LIN {X -0.062,Y -576.577,Z 1331.562,A 0.000,B 0.000,C 90.000,E1 137.229} C_DIS
LIN {X -0.112,Y -582.728,Z 1331.561,A 0.000,B 0.000,C 90.000,E1 136.905} C_DIS
LIN {X -0.019,Y -586.967,Z 1331.559,A 0.000,B 0.000,C 90.000,E1 136.620} C_DIS
LIN {X -0.228,Y -592.649,Z 1331.557,A 0.000,B 0.000,C 90.000,E1 136.215} C_DIS
LIN {X -0.386,Y -596.705,Z 1331.555,A 0.000,B 0.000,C 90.000,E1 135.891} C_DIS
LIN {X 0.112,Y -600.626,Z 1331.553,A 0.000,B 0.000,C 90.000,E1 135.486} C_DIS
LIN {X -0.001,Y -606.973,Z 1331.549,A 0.000,B 0.000,C 90.000,E1 134.879} C_DIS
LIN {X -0.167,Y -610.638,Z 1331.547,A 0.000,B 0.000,C 90.000,E1 134.514} C_DIS
LIN {X -0.298,Y -618.235,Z 1331.542,A 0.000,B 0.000,C 90.000,E1 133.623} C_DIS
LIN {X -0.305,Y -624.374,Z 1331.538,A 0.000,B 0.000,C 90.000,E1 132.852} C_DIS
LIN {X -0.246,Y -630.021,Z 1331.534,A 0.000,B 0.000,C 90.000,E1 132.081} C_DIS
LIN {X -0.360,Y -639.806,Z 1331.526,A 0.000,B 0.000,C 90.000,E1 130.701} C_DIS
LIN {X -0.233,Y -647.239,Z 1331.520,A 0.000,B 0.000,C 90.000,E1 129.564} C_DIS
LIN {X 0.131,Y -651.204,Z 1331.516,A 0.000,B 0.000,C 90.000,E1 128.910} C_DIS
LIN {X 0.016,Y -657.983,Z 1331.510,A 0.000,B 0.000,C 90.000,E1 127.810} C_DIS
LIN {X -0.050,Y -661.508,Z 1331.507,A 0.000,B 0.000,C 90.000,E1 127.202} C_DIS
LIN {X 0.091,Y -665.436,Z 1331.503,A 0.000,B 0.000,C 90.000,E1 126.457} C_DIS
LIN {X -0.320,Y -668.389,Z 1331.499,A 0.000,B 0.000,C 90.000,E1 125.884} C_DIS
LIN {X 0.287,Y -671.652,Z 1331.495,A 0.000,B 0.000,C 90.000,E1 125.105} C_DIS
LIN {X -0.155,Y -673.656,Z 1331.493,A 0.000,B 0.000,C 90.000,E1 124.659} C_DIS
LIN {X 0.118,Y -676.353,Z 1331.489,A 0.000,B 0.000,C 90.000,E1 123.913} C_DIS
LIN {X -0.143,Y -678.675,Z 1331.484,A 0.000,B 0.000,C 90.000,E1 123.214} C_DIS
LIN {X -0.205,Y -681.301,Z 1331.479,A 0.000,B 0.000,C 90.000,E1 122.260} C_DIS
LIN {X -0.208,Y -683.012,Z 1331.475,A 0.000,B 0.000,C 90.000,E1 121.544} C_DIS
LIN {X 0.166,Y -684.515,Z 1331.471,A 0.000,B 0.000,C 90.000,E1 120.797} C_DIS
LIN {X 0.207,Y -685.843,Z 1331.467,A 0.000,B 0.000,C 90.000,E1 120.079} C_DIS
LIN {X -0.333,Y -686.828,Z 1331.463,A 0.000,B 0.000,C 90.000,E1 119.411} C_DIS
LIN {X -0.267,Y -687.514,Z 1331.459,A 0.000,B 0.000,C 90.000,E1 118.693} C_DIS
LIN {X -0.193,Y -687.911,Z 1331.455,A 0.000,B 0.000,C 90.000,E1 117.975} C_DIS
LIN {X 0.110,Y -688.126,Z 1331.450,A 0.000,B 0.000,C 90.000,E1 117.001} C_DIS
LIN {X -0.124,Y -688.029,Z 1331.446,A 0.000,B 0.000,C 90.000,E1 116.309} C_DIS
LIN {X -0.282,Y -687.859,Z 1331.443,A 0.000,B 0.000,C 90.000,E1 115.848} C_DIS
LIN {X 0.173,Y -687.510,Z 1331.441,A 0.000,B 0.000,C 90.000,E1 115.335} C_DIS
LIN {X -0.064,Y -686.536,Z 1331.437,A 0.000,B 0.000,C 90.000,E1 114.643} C_DIS
LIN {X 0.097,Y -685.440,Z 1331.434,A 0.000,B 0.000,C 90.000,E1 114.155} C_DIS
LIN {X -0.309,Y -684.576,Z 1331.433,A 0.000,B 0.000,C 90.000,E1 113.951} C_DIS
LIN {X -0.155,Y -682.367,Z 1331.430,A 0.000,B 0.000,C 90.000,E1 113.462} C_DIS
LIN {X -0.051,Y -681.471,Z 1331.430,A 0.000,B 0.000,C 90.000,E1 113.334} C_DIS
LIN {X 0.357,Y -676.839,Z 1331.427,A 0.000,B 0.000,C 90.000,E1 112.823} C_DIS
LIN {X 0.189,Y -675.138,Z 1331.426,A 0.000,B 0.000,C 90.000,E1 112.717} C_DIS
LIN {X -0.013,Y -668.323,Z 1331.425,A 0.000,B 0.000,C 90.000,E1 112.408} C_DIS
LIN {X -0.068,Y -666.391,Z 1331.424,A 0.000,B 0.000,C 90.000,E1 112.333} C_DIS
LIN {X 0.000,Y -659.861,Z 1331.423,A 0.000,B 0.000,C 90.000,E1 112.153} C_DIS
LIN {X 0.072,Y -657.595,Z 1331.423,A 0.000,B 0.000,C 90.000,E1 112.099} C_DIS
LIN {X -0.013,Y -646.608,Z 1331.422,A 0.000,B 0.000,C 90.000,E1 111.950} C_DIS
LIN {X 0.023,Y -643.350,Z 1331.422,A 0.000,B 0.000,C 90.000,E1 111.897} C_DIS
LIN {X 0.052,Y -641.499,Z 1331.421,A 0.000,B 0.000,C 90.000,E1 111.844} C_DIS
LIN {X 0.018,Y -641.457,Z 1331.421,A 0.000,B 0.000,C 90.000,E1 111.844} C_DIS
LIN {X -0.197,Y -642.666,Z 1331.420,A 0.000,B 0.000,C 90.000,E1 111.663} C_DIS
LIN {X 0.238,Y -647.960,Z 1331.417,A 0.000,B 0.000,C 90.000,E1 110.972} C_DIS
LIN {X 0.157,Y -651.763,Z 1331.414,A 0.000,B 0.000,C 90.000,E1 110.482} C_DIS
LIN {X -0.079,Y -655.885,Z 1331.411,A 0.000,B 0.000,C 90.000,E1 109.885} C_DIS
LIN {X -0.057,Y -659.444,Z 1331.407,A 0.000,B 0.000,C 90.000,E1 109.268} C_DIS
LIN {X -0.226,Y -662.475,Z 1331.404,A 0.000,B 0.000,C 90.000,E1 108.671} C_DIS
LIN {X -0.313,Y -665.638,Z 1331.400,A 0.000,B 0.000,C 90.000,E1 107.946} C_DIS
LIN {X -0.373,Y -668.406,Z 1331.396,A 0.000,B 0.000,C 90.000,E1 107.221} C_DIS
LIN {X 0.306,Y -670.155,Z 1331.393,A 0.000,B 0.000,C 90.000,E1 106.677} C_DIS
LIN {X 0.098,Y -672.322,Z 1331.389,A 0.000,B 0.000,C 90.000,E1 105.969} C_DIS
LIN {X 0.155,Y -673.642,Z 1331.386,A 0.000,B 0.000,C 90.000,E1 105.481} C_DIS
LIN {X -0.019,Y -675.326,Z 1331.382,A 0.000,B 0.000,C 90.000,E1 104.773} C_DIS
LIN {X -0.124,Y -676.313,Z 1331.379,A 0.000,B 0.000,C 90.000,E1 104.300} C_DIS
LIN {X -0.270,Y -677.357,Z 1331.375,A 0.000,B 0.000,C 90.000,E1 103.592} C_DIS
LIN {X 0.299,Y -677.875,Z 1331.373,A 0.000,B 0.000,C 90.000,E1 103.063} C_DIS
LIN {X 0.121,Y -678.259,Z 1331.367,A 0.000,B 0.000,C 90.000,E1 102.119} C_DIS
LIN {X -0.151,Y -678.121,Z 1331.363,A 0.000,B 0.000,C 90.000,E1 101.422} C_DIS
LIN {X -0.243,Y -677.718,Z 1331.361,A 0.000,B 0.000,C 90.000,E1 100.950} C_DIS
LIN {X 0.152,Y -676.717,Z 1331.357,A 0.000,B 0.000,C 90.000,E1 100.197} C_DIS
LIN {X 0.045,Y -675.836,Z 1331.354,A 0.000,B 0.000,C 90.000,E1 99.726} C_DIS
LIN {X -0.183,Y -674.676,Z 1331.351,A 0.000,B 0.000,C 90.000,E1 99.265} C_DIS
LIN {X 0.251,Y -673.113,Z 1331.349,A 0.000,B 0.000,C 90.000,E1 98.746} C_DIS
LIN {X -0.061,Y -670.258,Z 1331.345,A 0.000,B 0.000,C 90.000,E1 98.049} C_DIS
LIN {X -0.313,Y -668.104,Z 1331.342,A 0.000,B 0.000,C 90.000,E1 97.587} C_DIS
LIN {X -0.107,Y -663.890,Z 1331.337,A 0.000,B 0.000,C 90.000,E1 96.720} C_DIS
LIN {X 0.135,Y -659.920,Z 1331.333,A 0.000,B 0.000,C 90.000,E1 95.967} C_DIS
LIN {X -0.253,Y -656.964,Z 1331.331,A 0.000,B 0.000,C 90.000,E1 95.511} C_DIS
LIN {X -0.039,Y -652.848,Z 1331.327,A 0.000,B 0.000,C 90.000,E1 94.878} C_DIS
LIN {X 0.135,Y -648.411,Z 1331.324,A 0.000,B 0.000,C 90.000,E1 94.245} C_DIS
LIN {X -0.262,Y -644.634,Z 1331.321,A 0.000,B 0.000,C 90.000,E1 93.784} C_DIS
LIN {X 0.038,Y -641.655,Z 1331.319,A 0.000,B 0.000,C 90.000,E1 93.383} C_DIS
LIN {X 0.109,Y -636.035,Z 1331.315,A 0.000,B 0.000,C 90.000,E1 92.751} C_DIS
LIN {X 0.212,Y -629.898,Z 1331.312,A 0.000,B 0.000,C 90.000,E1 92.121} C_DIS
LIN {X 0.185,Y -619.842,Z 1331.307,A 0.000,B 0.000,C 90.000,E1 91.146} C_DIS
LIN {X -0.039,Y -615.737,Z 1331.304,A 0.000,B 0.000,C 90.000,E1 90.802} C_DIS
LIN {X -0.001,Y -610.127,Z 1331.302,A 0.000,B 0.000,C 90.000,E1 90.344} C_DIS
LIN {X 0.018,Y -608.545,Z 1331.301,A 0.000,B 0.000,C 90.000,E1 90.229} C_DIS
LIN {X 0.053,Y -602.004,Z 1331.299,A 0.000,B 0.000,C 90.000,E1 89.828} C_DIS
LIN {X -0.038,Y -594.968,Z 1331.297,A 0.000,B 0.000,C 90.000,E1 89.484} C_DIS
LIN {X -0.226,Y -587.786,Z 1331.296,A 0.000,B 0.000,C 90.000,E1 89.198} C_DIS
LIN {X -0.262,Y -577.938,Z 1331.293,A 0.000,B 0.000,C 90.000,E1 88.797} C_DIS
LIN {X 0.160,Y -576.610,Z 1331.293,A 0.000,B 0.000,C 90.000,E1 88.682} C_DIS
LIN {X 0.074,Y -573.479,Z 1331.292,A 0.000,B 0.000,C 90.000,E1 88.453} C_DIS
LIN {X 0.131,Y -573.050,Z 1331.291,A 0.000,B 0.000,C 90.000,E1 88.396} C_DIS
LIN {X 0.097,Y -573.038,Z 1331.291,A 0.000,B 0.000,C 90.000,E1 88.396} C_DIS
LIN {X 0.284,Y -572.281,Z 1331.290,A 0.000,B 0.000,C 90.000,E1 88.108} C_DIS
LIN {X 0.249,Y -572.134,Z 1331.287,A 0.000,B 0.000,C 90.000,E1 87.650} C_DIS
LIN {X 0.140,Y -574.875,Z 1331.271,A 0.000,B 0.000,C 90.000,E1 84.666} C_DIS
LIN {X -0.183,Y -577.423,Z 1331.258,A 0.000,B 0.000,C 90.000,E1 82.527} C_DIS
LIN {X -0.207,Y -579.382,Z 1331.249,A 0.000,B 0.000,C 90.000,E1 80.905} C_DIS
LIN {X -0.097,Y -581.262,Z 1331.240,A 0.000,B 0.000,C 90.000,E1 79.275} C_DIS
LIN {X -0.192,Y -582.690,Z 1331.233,A 0.000,B 0.000,C 90.000,E1 77.937} C_DIS
LIN {X 0.084,Y -584.057,Z 1331.224,A 0.000,B 0.000,C 90.000,E1 76.297} C_DIS
LIN {X 0.042,Y -584.865,Z 1331.218,A 0.000,B 0.000,C 90.000,E1 75.227} C_DIS
LIN {X -0.233,Y -586.188,Z 1331.208,A 0.000,B 0.000,C 90.000,E1 73.378} C_DIS
LIN {X -0.160,Y -587.169,Z 1331.199,A 0.000,B 0.000,C 90.000,E1 71.764} C_DIS
LIN {X 0.106,Y -588.256,Z 1331.190,A 0.000,B 0.000,C 90.000,E1 70.134} C_DIS
LIN {X -0.197,Y -589.629,Z 1331.178,A 0.000,B 0.000,C 90.000,E1 68.028} C_DIS
LIN {X 0.088,Y -591.002,Z 1331.166,A 0.000,B 0.000,C 90.000,E1 65.869} C_DIS
LIN {X 0.208,Y -591.781,Z 1331.160,A 0.000,B 0.000,C 90.000,E1 64.793} C_DIS
LIN {X 0.044,Y -593.113,Z 1331.150,A 0.000,B 0.000,C 90.000,E1 62.948} C_DIS
LIN {X -0.060,Y -594.629,Z 1331.140,A 0.000,B 0.000,C 90.000,E1 61.101} C_DIS
LIN {X -0.108,Y -596.409,Z 1331.129,A 0.000,B 0.000,C 90.000,E1 59.253} C_DIS
LIN {X 0.188,Y -598.296,Z 1331.119,A 0.000,B 0.000,C 90.000,E1 57.375} C_DIS
LIN {X -0.133,Y -599.720,Z 1331.112,A 0.000,B 0.000,C 90.000,E1 56.087} C_DIS
LIN {X -0.101,Y -601.081,Z 1331.104,A 0.000,B 0.000,C 90.000,E1 54.769} C_DIS
LIN {X 0.216,Y -603.046,Z 1331.093,A 0.000,B 0.000,C 90.000,E1 52.637} C_DIS
LIN {X 0.171,Y -603.992,Z 1331.085,A 0.000,B 0.000,C 90.000,E1 51.331} C_DIS
LIN {X 0.058,Y -604.891,Z 1331.078,A 0.000,B 0.000,C 90.000,E1 50.033} C_DIS
LIN {X -0.225,Y -605.436,Z 1331.072,A 0.000,B 0.000,C 90.000,E1 49.013} C_DIS
LIN {X -0.114,Y -605.758,Z 1331.066,A 0.000,B 0.000,C 90.000,E1 47.957} C_DIS
LIN {X -0.176,Y -606.045,Z 1331.056,A 0.000,B 0.000,C 90.000,E1 46.134} C_DIS
LIN {X -0.084,Y -606.096,Z 1331.050,A 0.000,B 0.000,C 90.000,E1 45.081} C_DIS
LIN {X 0.008,Y -605.920,Z 1331.045,A 0.000,B 0.000,C 90.000,E1 44.028} C_DIS
LIN {X -0.130,Y -605.679,Z 1331.040,A 0.000,B 0.000,C 90.000,E1 43.257} C_DIS
LIN {X 0.198,Y -605.220,Z 1331.033,A 0.000,B 0.000,C 90.000,E1 41.919} C_DIS
LIN {X -0.094,Y -604.592,Z 1331.024,A 0.000,B 0.000,C 90.000,E1 40.378} C_DIS
LIN {X -0.332,Y -603.783,Z 1331.016,A 0.000,B 0.000,C 90.000,E1 38.830} C_DIS
LIN {X -0.033,Y -603.330,Z 1331.011,A 0.000,B 0.000,C 90.000,E1 38.016} C_DIS
LIN {X 0.147,Y -602.529,Z 1331.005,A 0.000,B 0.000,C 90.000,E1 36.950} C_DIS
LIN {X -0.168,Y -601.163,Z 1331.000,A 0.000,B 0.000,C 90.000,E1 35.931} C_DIS
LIN {X 0.225,Y -599.928,Z 1330.995,A 0.000,B 0.000,C 90.000,E1 35.105} C_DIS
LIN {X 0.016,Y -598.152,Z 1330.989,A 0.000,B 0.000,C 90.000,E1 34.072} C_DIS
LIN {X -0.344,Y -597.115,Z 1330.986,A 0.000,B 0.000,C 90.000,E1 33.579} C_DIS
LIN {X 0.127,Y -594.080,Z 1330.979,A 0.000,B 0.000,C 90.000,E1 32.212} C_DIS
LIN {X 0.237,Y -592.668,Z 1330.976,A 0.000,B 0.000,C 90.000,E1 31.671} C_DIS
LIN {X -0.388,Y -589.347,Z 1330.970,A 0.000,B 0.000,C 90.000,E1 30.669} C_DIS
LIN {X 0.082,Y -586.485,Z 1330.966,A 0.000,B 0.000,C 90.000,E1 29.823} C_DIS
LIN {X 0.135,Y -584.367,Z 1330.963,A 0.000,B 0.000,C 90.000,E1 29.283} C_DIS
LIN {X 0.039,Y -580.809,Z 1330.958,A 0.000,B 0.000,C 90.000,E1 28.487} C_DIS
LIN {X -0.228,Y -578.276,Z 1330.955,A 0.000,B 0.000,C 90.000,E1 27.975} C_DIS
LIN {X 0.112,Y -574.080,Z 1330.951,A 0.000,B 0.000,C 90.000,E1 27.129} C_DIS
LIN {X -0.283,Y -570.240,Z 1330.947,A 0.000,B 0.000,C 90.000,E1 26.488} C_DIS
LIN {X -0.196,Y -566.070,Z 1330.943,A 0.000,B 0.000,C 90.000,E1 25.796} C_DIS
LIN {X 0.191,Y -562.510,Z 1330.940,A 0.000,B 0.000,C 90.000,E1 25.207} C_DIS
LIN {X 0.307,Y -558.636,Z 1330.937,A 0.000,B 0.000,C 90.000,E1 24.643} C_DIS
LIN {X 0.062,Y -551.462,Z 1330.932,A 0.000,B 0.000,C 90.000,E1 23.695} C_DIS
LIN {X 0.143,Y -544.586,Z 1330.927,A 0.000,B 0.000,C 90.000,E1 22.845} C_DIS
LIN {X -0.216,Y -538.717,Z 1330.923,A 0.000,B 0.000,C 90.000,E1 22.206} C_DIS
LIN {X 0.226,Y -533.817,Z 1330.920,A 0.000,B 0.000,C 90.000,E1 21.589} C_DIS
LIN {X 0.072,Y -523.295,Z 1330.914,A 0.000,B 0.000,C 90.000,E1 20.482} C_DIS
LIN {X -0.222,Y -512.601,Z 1330.908,A 0.000,B 0.000,C 90.000,E1 19.396} C_DIS
LIN {X 0.248,Y -503.297,Z 1330.902,A 0.000,B 0.000,C 90.000,E1 18.362} C_DIS
LIN {X 0.005,Y -492.422,Z 1330.896,A 0.000,B 0.000,C 90.000,E1 17.330} C_DIS
LIN {X 0.045,Y -478.128,Z 1330.889,A 0.000,B 0.000,C 90.000,E1 15.969} C_DIS
LIN {X 0.080,Y -468.016,Z 1330.884,A 0.000,B 0.000,C 90.000,E1 15.009} C_DIS
LIN {X 0.147,Y -451.951,Z 1330.875,A 0.000,B 0.000,C 90.000,E1 13.480} C_DIS
LIN {X -0.018,Y -431.896,Z 1330.864,A 0.000,B 0.000,C 90.000,E1 11.478} C_DIS
LIN {X -0.191,Y -417.628,Z 1330.855,A 0.000,B 0.000,C 90.000,E1 9.962} C_DIS
LIN {X -0.042,Y -404.851,Z 1330.847,A 0.000,B 0.000,C 90.000,E1 8.511} C_DIS
LIN {X -0.076,Y -399.255,Z 1330.844,A 0.000,B 0.000,C 90.000,E1 7.871} C_DIS
LIN {X -0.072,Y -395.398,Z 1330.841,A 0.000,B 0.000,C 90.000,E1 7.352} C_DIS
LIN {X 0.017,Y -395.218,Z 1330.841,A 0.000,B 0.000,C 90.000,E1 7.296} C_DIS
LIN {X -0.020,Y -395.210,Z 1330.841,A 0.000,B 0.000,C 90.000,E1 7.296} C_DIS
LIN {X 0.119,Y -395.467,Z 1330.840,A 0.000,B 0.000,C 90.000,E1 7.182} C_DIS
LIN {X 0.081,Y -395.514,Z 1330.840,A 0.000,B 0.000,C 90.000,E1 7.182} C_DIS
LIN {X 0.073,Y -398.573,Z 1330.838,A 0.000,B 0.000,C 90.000,E1 6.891} C_DIS
LIN {X -0.153,Y -400.282,Z 1330.838,A 0.000,B 0.000,C 90.000,E1 6.777} C_DIS
LIN {X 0.049,Y -413.967,Z 1330.833,A 0.000,B 0.000,C 90.000,E1 5.853} C_DIS
LIN {X 0.107,Y -417.244,Z 1330.831,A 0.000,B 0.000,C 90.000,E1 5.625} C_DIS
LIN {X -0.069,Y -425.051,Z 1330.828,A 0.000,B 0.000,C 90.000,E1 5.049} C_DIS
LIN {X 0.062,Y -429.652,Z 1330.826,A 0.000,B 0.000,C 90.000,E1 4.645} C_DIS
LIN {X -0.137,Y -438.664,Z 1330.821,A 0.000,B 0.000,C 90.000,E1 3.841} C_DIS
LIN {X 0.072,Y -445.876,Z 1330.817,A 0.000,B 0.000,C 90.000,E1 3.094} C_DIS
LIN {X 0.057,Y -452.935,Z 1330.813,A 0.000,B 0.000,C 90.000,E1 2.350} C_DIS
LIN {X -0.061,Y -459.618,Z 1330.809,A 0.000,B 0.000,C 90.000,E1 1.604} C_DIS
LIN {X 0.202,Y -465.898,Z 1330.805,A 0.000,B 0.000,C 90.000,E1 0.802} C_DIS
LIN {X 0.191,Y -470.762,Z 1330.801,A 0.000,B 0.000,C 90.000,E1 0.172} C_DIS
LIN {X 0.093,Y -476.831,Z 1330.796,A 0.000,B 0.000,C 90.000,E1 359.312} C_DIS
LIN {X -0.177,Y -481.811,Z 1330.792,A 0.000,B 0.000,C 90.000,E1 358.568} C_DIS
LIN {X 0.100,Y -486.338,Z 1330.788,A 0.000,B 0.000,C 90.000,E1 357.764} C_DIS
LIN {X -0.087,Y -490.693,Z 1330.783,A 0.000,B 0.000,C 90.000,E1 357.020} C_DIS
LIN {X 0.112,Y -493.901,Z 1330.780,A 0.000,B 0.000,C 90.000,E1 356.388} C_DIS
LIN {X 0.022,Y -497.559,Z 1330.776,A 0.000,B 0.000,C 90.000,E1 355.641} C_DIS
LIN {X 0.146,Y -501.640,Z 1330.771,A 0.000,B 0.000,C 90.000,E1 354.723} C_DIS
LIN {X 0.123,Y -504.809,Z 1330.767,A 0.000,B 0.000,C 90.000,E1 353.976} C_DIS
LIN {X -0.010,Y -507.132,Z 1330.763,A 0.000,B 0.000,C 90.000,E1 353.394} C_DIS
LIN {X 0.157,Y -511.513,Z 1330.757,A 0.000,B 0.000,C 90.000,E1 352.186} C_DIS
LIN {X 0.081,Y -513.454,Z 1330.753,A 0.000,B 0.000,C 90.000,E1 351.602} C_DIS
LIN {X -0.100,Y -516.862,Z 1330.747,A 0.000,B 0.000,C 90.000,E1 350.443} C_DIS
LIN {X -0.138,Y -519.199,Z 1330.742,A 0.000,B 0.000,C 90.000,E1 349.567} C_DIS
LIN {X -0.249,Y -521.216,Z 1330.737,A 0.000,B 0.000,C 90.000,E1 348.701} C_DIS
LIN {X -0.133,Y -523.042,Z 1330.732,A 0.000,B 0.000,C 90.000,E1 347.813} C_DIS
LIN {X -0.090,Y -525.127,Z 1330.726,A 0.000,B 0.000,C 90.000,E1 346.645} C_DIS
LIN {X -0.062,Y -526.045,Z 1330.723,A 0.000,B 0.000,C 90.000,E1 346.061} C_DIS
LIN {X 0.117,Y -527.163,Z 1330.718,A 0.000,B 0.000,C 90.000,E1 345.172} C_DIS
LIN {X -0.198,Y -528.147,Z 1330.713,A 0.000,B 0.000,C 90.000,E1 344.338} C_DIS
LIN {X 0.004,Y -528.829,Z 1330.708,A 0.000,B 0.000,C 90.000,E1 343.449} C_DIS
LIN {X 0.192,Y -529.155,Z 1330.705,A 0.000,B 0.000,C 90.000,E1 342.851} C_DIS
LIN {X 0.068,Y -529.356,Z 1330.698,A 0.000,B 0.000,C 90.000,E1 341.710} C_DIS
LIN {X -0.065,Y -529.297,Z 1330.694,A 0.000,B 0.000,C 90.000,E1 340.859} C_DIS
LIN {X 0.300,Y -528.995,Z 1330.690,A 0.000,B 0.000,C 90.000,E1 340.242} C_DIS
LIN {X -0.145,Y -528.127,Z 1330.684,A 0.000,B 0.000,C 90.000,E1 339.135} C_DIS
LIN {X 0.203,Y -526.930,Z 1330.679,A 0.000,B 0.000,C 90.000,E1 338.230} C_DIS
LIN {X 0.093,Y -524.425,Z 1330.671,A 0.000,B 0.000,C 90.000,E1 336.794} C_DIS
LIN {X 0.103,Y -522.563,Z 1330.666,A 0.000,B 0.000,C 90.000,E1 335.921} C_DIS
LIN {X 0.089,Y -520.368,Z 1330.661,A 0.000,B 0.000,C 90.000,E1 335.049} C_DIS
LIN {X -0.061,Y -516.851,Z 1330.655,A 0.000,B 0.000,C 90.000,E1 333.896} C_DIS
LIN {X 0.090,Y -512.241,Z 1330.647,A 0.000,B 0.000,C 90.000,E1 332.410} C_DIS
LIN {X 0.182,Y -509.383,Z 1330.642,A 0.000,B 0.000,C 90.000,E1 331.513} C_DIS
LIN {X -0.028,Y -506.591,Z 1330.638,A 0.000,B 0.000,C 90.000,E1 330.795} C_DIS
LIN {X 0.109,Y -504.527,Z 1330.635,A 0.000,B 0.000,C 90.000,E1 330.333} C_DIS
LIN {X -0.014,Y -502.929,Z 1330.634,A 0.000,B 0.000,C 90.000,E1 330.049} C_DIS
LIN {X 0.041,Y -500.988,Z 1330.632,A 0.000,B 0.000,C 90.000,E1 329.744} C_DIS
LIN {X -0.151,Y -499.776,Z 1330.631,A 0.000,B 0.000,C 90.000,E1 329.616} C_DIS
LIN {X -0.090,Y -498.041,Z 1330.630,A 0.000,B 0.000,C 90.000,E1 329.459} C_DIS
LIN {X -0.222,Y -472.486,Z 1330.620,A 0.000,B 0.000,C 90.000,E1 327.661} C_DIS
LIN {X -0.018,Y -449.591,Z 1330.610,A 0.000,B 0.000,C 90.000,E1 325.801} C_DIS
LIN {X 0.050,Y -428.701,Z 1330.600,A 0.000,B 0.000,C 90.000,E1 323.909} C_DIS
LIN {X 0.168,Y -408.338,Z 1330.588,A 0.000,B 0.000,C 90.000,E1 321.823} C_DIS
LIN {X -0.045,Y -389.975,Z 1330.576,A 0.000,B 0.000,C 90.000,E1 319.747} C_DIS
LIN {X 0.005,Y -377.260,Z 1330.567,A 0.000,B 0.000,C 90.000,E1 318.119} C_DIS
LIN {X 0.219,Y -377.263,Z 1330.567,A 0.000,B 0.000,C 90.000,E1 318.081} C_DIS
LIN {X -0.089,Y -377.906,Z 1330.565,A 0.000,B 0.000,C 90.000,E1 317.634} C_DIS
LIN {X -0.082,Y -378.509,Z 1330.561,A 0.000,B 0.000,C 90.000,E1 316.905} C_DIS
LIN {X 0.218,Y -384.511,Z 1330.528,A 0.000,B 0.000,C 90.000,E1 311.067} C_DIS
LIN {X -0.029,Y -384.928,Z 1330.526,A 0.000,B 0.000,C 90.000,E1 310.744} C_DIS
LIN {X -0.109,Y -390.684,Z 1330.495,A 0.000,B 0.000,C 90.000,E1 305.025} C_DIS
LIN {X -0.042,Y -391.181,Z 1330.493,A 0.000,B 0.000,C 90.000,E1 304.659} C_DIS
LIN {X 0.086,Y -396.896,Z 1330.459,A 0.000,B 0.000,C 90.000,E1 298.615} C_DIS
LIN {X -0.137,Y -397.492,Z 1330.453,A 0.000,B 0.000,C 90.000,E1 297.590} C_DIS
LIN {X 0.096,Y -401.633,Z 1330.426,A 0.000,B 0.000,C 90.000,E1 292.642} C_DIS
LIN {X -0.153,Y -404.705,Z 1330.395,A 0.000,B 0.000,C 90.000,E1 287.094} C_DIS
LIN {X -0.161,Y -406.131,Z 1330.364,A 0.000,B 0.000,C 90.000,E1 281.535} C_DIS
LIN {X -0.118,Y -405.722,Z 1330.356,A 0.000,B 0.000,C 90.000,E1 280.141} C_DIS
LIN {X -0.068,Y -405.689,Z 1330.333,A 0.000,B 0.000,C 90.000,E1 275.967} C_DIS
LIN {X -0.031,Y -403.464,Z 1330.304,A 0.000,B 0.000,C 90.000,E1 270.745} C_DIS
LIN {X -0.063,Y -403.248,Z 1330.302,A 0.000,B 0.000,C 90.000,E1 270.401} C_DIS
LIN {X 0.116,Y -398.868,Z 1330.271,A 0.000,B 0.000,C 90.000,E1 264.780} C_DIS
LIN {X 0.014,Y -393.344,Z 1330.244,A 0.000,B 0.000,C 90.000,E1 259.859} C_DIS
LIN {X -0.064,Y -392.771,Z 1330.240,A 0.000,B 0.000,C 90.000,E1 259.162} C_DIS
LIN {X 0.015,Y -386.319,Z 1330.214,A 0.000,B 0.000,C 90.000,E1 254.519} C_DIS
LIN {X -0.024,Y -385.215,Z 1330.208,A 0.000,B 0.000,C 90.000,E1 253.449} C_DIS
LIN {X 0.017,Y -384.010,Z 1330.204,A 0.000,B 0.000,C 90.000,E1 252.725} C_DIS
LIN {X -0.154,Y -377.445,Z 1330.180,A 0.000,B 0.000,C 90.000,E1 248.411} C_DIS
LIN {X -0.062,Y -376.171,Z 1330.174,A 0.000,B 0.000,C 90.000,E1 247.305} C_DIS
LIN {X -0.073,Y -368.341,Z 1330.147,A 0.000,B 0.000,C 90.000,E1 242.538} C_DIS
LIN {X -0.030,Y -366.478,Z 1330.139,A 0.000,B 0.000,C 90.000,E1 241.051} C_DIS
LIN {X 0.055,Y -365.937,Z 1330.137,A 0.000,B 0.000,C 90.000,E1 240.667} C_DIS
LIN {X -0.055,Y -359.116,Z 1330.114,A 0.000,B 0.000,C 90.000,E1 236.580} C_DIS
LIN {X -0.059,Y -356.258,Z 1330.102,A 0.000,B 0.000,C 90.000,E1 234.322} C_DIS
LIN {X 0.161,Y -355.737,Z 1330.100,A 0.000,B 0.000,C 90.000,E1 233.909} C_DIS
LIN {X -0.036,Y -348.721,Z 1330.074,A 0.000,B 0.000,C 90.000,E1 229.380} C_DIS
LIN {X -0.126,Y -346.015,Z 1330.061,A 0.000,B 0.000,C 90.000,E1 226.986} C_DIS
LIN {X -0.144,Y -346.013,Z 1330.061,A 0.000,B 0.000,C 90.000,E1 226.986} C_DIS
LIN {X -0.006,Y -360.672,Z 1330.048,A 0.000,B 0.000,C 90.000,E1 224.595} C_DIS
LIN {X 0.129,Y -377.606,Z 1330.034,A 0.000,B 0.000,C 90.000,E1 222.162} C_DIS
LIN {X 0.014,Y -395.894,Z 1330.022,A 0.000,B 0.000,C 90.000,E1 219.886} C_DIS
LIN {X -0.121,Y -414.801,Z 1330.010,A 0.000,B 0.000,C 90.000,E1 217.810} C_DIS
LIN {X 0.112,Y -435.728,Z 1329.999,A 0.000,B 0.000,C 90.000,E1 215.724} C_DIS
LIN {X 0.210,Y -443.323,Z 1329.995,A 0.000,B 0.000,C 90.000,E1 215.025} C_DIS
LIN {X 0.145,Y -444.425,Z 1329.994,A 0.000,B 0.000,C 90.000,E1 214.898} C_DIS
LIN {X 0.115,Y -445.341,Z 1329.993,A 0.000,B 0.000,C 90.000,E1 214.739} C_DIS
LIN {X -0.170,Y -446.067,Z 1329.992,A 0.000,B 0.000,C 90.000,E1 214.612} C_DIS
LIN {X -0.111,Y -447.221,Z 1329.990,A 0.000,B 0.000,C 90.000,E1 214.278} C_DIS
LIN {X -0.102,Y -448.948,Z 1329.987,A 0.000,B 0.000,C 90.000,E1 213.627} C_DIS
LIN {X 0.046,Y -450.265,Z 1329.983,A 0.000,B 0.000,C 90.000,E1 212.959} C_DIS
LIN {X -0.087,Y -451.657,Z 1329.978,A 0.000,B 0.000,C 90.000,E1 212.005} C_DIS
LIN {X 0.071,Y -453.767,Z 1329.967,A 0.000,B 0.000,C 90.000,E1 210.050} C_DIS
LIN {X -0.194,Y -457.672,Z 1329.949,A 0.000,B 0.000,C 90.000,E1 206.873} C_DIS
LIN {X 0.090,Y -461.390,Z 1329.935,A 0.000,B 0.000,C 90.000,E1 204.283} C_DIS
LIN {X 0.008,Y -463.949,Z 1329.924,A 0.000,B 0.000,C 90.000,E1 202.386} C_DIS
LIN {X 0.109,Y -466.055,Z 1329.916,A 0.000,B 0.000,C 90.000,E1 200.791} C_DIS
LIN {X 0.151,Y -467.669,Z 1329.909,A 0.000,B 0.000,C 90.000,E1 199.523} C_DIS
LIN {X 0.174,Y -469.639,Z 1329.900,A 0.000,B 0.000,C 90.000,E1 197.946} C_DIS
LIN {X 0.087,Y -471.642,Z 1329.891,A 0.000,B 0.000,C 90.000,E1 196.386} C_DIS
LIN {X -0.145,Y -473.804,Z 1329.881,A 0.000,B 0.000,C 90.000,E1 194.537} C_DIS
LIN {X 0.003,Y -475.988,Z 1329.870,A 0.000,B 0.000,C 90.000,E1 192.647} C_DIS
LIN {X -0.154,Y -478.570,Z 1329.858,A 0.000,B 0.000,C 90.000,E1 190.489} C_DIS
LIN {X 0.047,Y -480.365,Z 1329.850,A 0.000,B 0.000,C 90.000,E1 188.916} C_DIS
LIN {X -0.130,Y -481.757,Z 1329.843,A 0.000,B 0.000,C 90.000,E1 187.701} C_DIS
LIN {X -0.010,Y -483.225,Z 1329.834,A 0.000,B 0.000,C 90.000,E1 186.144} C_DIS
LIN {X 0.136,Y -484.546,Z 1329.826,A 0.000,B 0.000,C 90.000,E1 184.588} C_DIS
LIN {X -0.197,Y -485.037,Z 1329.822,A 0.000,B 0.000,C 90.000,E1 184.012} C_DIS
LIN {X -0.225,Y -485.525,Z 1329.817,A 0.000,B 0.000,C 90.000,E1 183.094} C_DIS
LIN {X -0.113,Y -486.145,Z 1329.809,A 0.000,B 0.000,C 90.000,E1 181.547} C_DIS
LIN {X -0.143,Y -486.385,Z 1329.803,A 0.000,B 0.000,C 90.000,E1 180.630} C_DIS
LIN {X -0.021,Y -486.448,Z 1329.795,A 0.000,B 0.000,C 90.000,E1 179.083} C_DIS
LIN {X -0.034,Y -486.262,Z 1329.790,A 0.000,B 0.000,C 90.000,E1 178.165} C_DIS
LIN {X -0.239,Y -485.760,Z 1329.783,A 0.000,B 0.000,C 90.000,E1 176.963} C_DIS
LIN {X 0.080,Y -484.844,Z 1329.776,A 0.000,B 0.000,C 90.000,E1 175.698} C_DIS
LIN {X 0.238,Y -484.268,Z 1329.773,A 0.000,B 0.000,C 90.000,E1 175.065} C_DIS
LIN {X 0.058,Y -482.744,Z 1329.766,A 0.000,B 0.000,C 90.000,E1 173.856} C_DIS
LIN {X -0.149,Y -480.686,Z 1329.759,A 0.000,B 0.000,C 90.000,E1 172.648} C_DIS
LIN {X 0.035,Y -479.472,Z 1329.756,A 0.000,B 0.000,C 90.000,E1 172.008} C_DIS
LIN {X -0.180,Y -478.777,Z 1329.754,A 0.000,B 0.000,C 90.000,E1 171.724} C_DIS
LIN {X -0.160,Y -476.205,Z 1329.749,A 0.000,B 0.000,C 90.000,E1 170.792} C_DIS
LIN {X -0.005,Y -474.359,Z 1329.745,A 0.000,B 0.000,C 90.000,E1 170.151} C_DIS
LIN {X -0.055,Y -472.504,Z 1329.743,A 0.000,B 0.000,C 90.000,E1 169.690} C_DIS
LIN {X 0.255,Y -469.109,Z 1329.738,A 0.000,B 0.000,C 90.000,E1 168.870} C_DIS
LIN {X -0.108,Y -465.611,Z 1329.735,A 0.000,B 0.000,C 90.000,E1 168.285} C_DIS
LIN {X -0.040,Y -461.752,Z 1329.731,A 0.000,B 0.000,C 90.000,E1 167.645} C_DIS
LIN {X -0.187,Y -452.714,Z 1329.723,A 0.000,B 0.000,C 90.000,E1 166.228} C_DIS
LIN {X 0.223,Y -441.329,Z 1329.714,A 0.000,B 0.000,C 90.000,E1 164.393} C_DIS
LIN {X 0.026,Y -434.313,Z 1329.707,A 0.000,B 0.000,C 90.000,E1 163.268} C_DIS
LIN {X 0.253,Y -430.222,Z 1329.703,A 0.000,B 0.000,C 90.000,E1 162.417} C_DIS
LIN {X 0.101,Y -429.266,Z 1329.701,A 0.000,B 0.000,C 90.000,E1 162.127} C_DIS
LIN {X 0.013,Y -428.042,Z 1329.698,A 0.000,B 0.000,C 90.000,E1 161.638} C_DIS
LIN {X -0.027,Y -428.542,Z 1329.695,A 0.000,B 0.000,C 90.000,E1 161.094} C_DIS
LIN {X -0.067,Y -428.575,Z 1329.695,A 0.000,B 0.000,C 90.000,E1 161.094} C_DIS
LIN {X 0.127,Y -430.306,Z 1329.693,A 0.000,B 0.000,C 90.000,E1 160.786} C_DIS
LIN {X -0.091,Y -434.443,Z 1329.691,A 0.000,B 0.000,C 90.000,E1 160.423} C_DIS
LIN {X 0.235,Y -444.010,Z 1329.687,A 0.000,B 0.000,C 90.000,E1 159.571} C_DIS
LIN {X -0.257,Y -459.659,Z 1329.680,A 0.000,B 0.000,C 90.000,E1 158.411} C_DIS
LIN {X 0.060,Y -472.089,Z 1329.675,A 0.000,B 0.000,C 90.000,E1 157.411} C_DIS
LIN {X 0.169,Y -481.096,Z 1329.671,A 0.000,B 0.000,C 90.000,E1 156.666} C_DIS
LIN {X -0.036,Y -486.956,Z 1329.668,A 0.000,B 0.000,C 90.000,E1 156.177} C_DIS
LIN {X 0.104,Y -495.563,Z 1329.663,A 0.000,B 0.000,C 90.000,E1 155.357} C_DIS
LIN {X 0.144,Y -502.403,Z 1329.659,A 0.000,B 0.000,C 90.000,E1 154.665} C_DIS
LIN {X -0.228,Y -508.832,Z 1329.656,A 0.000,B 0.000,C 90.000,E1 154.024} C_DIS
LIN {X -0.105,Y -513.933,Z 1329.652,A 0.000,B 0.000,C 90.000,E1 153.435} C_DIS
LIN {X -0.167,Y -517.651,Z 1329.650,A 0.000,B 0.000,C 90.000,E1 152.999} C_DIS
LIN {X 0.025,Y -521.180,Z 1329.647,A 0.000,B 0.000,C 90.000,E1 152.538} C_DIS
LIN {X -0.163,Y -525.314,Z 1329.644,A 0.000,B 0.000,C 90.000,E1 151.975} C_DIS
LIN {X -0.078,Y -528.931,Z 1329.641,A 0.000,B 0.000,C 90.000,E1 151.385} C_DIS
LIN {X -0.112,Y -532.647,Z 1329.637,A 0.000,B 0.000,C 90.000,E1 150.667} C_DIS
LIN {X 0.149,Y -535.542,Z 1329.633,A 0.000,B 0.000,C 90.000,E1 149.921} C_DIS
LIN {X 0.312,Y -537.482,Z 1329.630,A 0.000,B 0.000,C 90.000,E1 149.331} C_DIS
LIN {X -0.255,Y -539.925,Z 1329.625,A 0.000,B 0.000,C 90.000,E1 148.535} C_DIS
LIN {X -0.055,Y -542.022,Z 1329.620,A 0.000,B 0.000,C 90.000,E1 147.661} C_DIS
LIN {X -0.018,Y -543.228,Z 1329.617,A 0.000,B 0.000,C 90.000,E1 147.089} C_DIS
LIN {X -0.053,Y -545.253,Z 1329.611,A 0.000,B 0.000,C 90.000,E1 145.960} C_DIS
LIN {X 0.055,Y -546.416,Z 1329.606,A 0.000,B 0.000,C 90.000,E1 145.102} C_DIS
LIN {X -0.091,Y -547.578,Z 1329.600,A 0.000,B 0.000,C 90.000,E1 143.989} C_DIS
LIN {X 0.099,Y -548.452,Z 1329.594,A 0.000,B 0.000,C 90.000,E1 142.844} C_DIS
LIN {X 0.024,Y -549.713,Z 1329.583,A 0.000,B 0.000,C 90.000,E1 140.884} C_DIS
LIN {X 0.214,Y -550.873,Z 1329.575,A 0.000,B 0.000,C 90.000,E1 139.461} C_DIS
LIN {X -0.098,Y -551.833,Z 1329.572,A 0.000,B 0.000,C 90.000,E1 138.933} C_DIS
LIN {X 0.068,Y -551.937,Z 1329.571,A 0.000,B 0.000,C 90.000,E1 138.771} C_DIS
LIN {X 0.026,Y -551.959,Z 1329.571,A 0.000,B 0.000,C 90.000,E1 138.771} C_DIS
LIN {X 0.166,Y -554.320,Z 1329.569,A 0.000,B 0.000,C 90.000,E1 138.485} C_DIS
LIN {X 0.272,Y -555.217,Z 1329.569,A 0.000,B 0.000,C 90.000,E1 138.405} C_DIS
LIN {X -0.037,Y -556.413,Z 1329.569,A 0.000,B 0.000,C 90.000,E1 138.366} C_DIS
LIN {X 0.032,Y -563.752,Z 1329.568,A 0.000,B 0.000,C 90.000,E1 138.162} C_DIS
LIN {X -0.148,Y -567.309,Z 1329.567,A 0.000,B 0.000,C 90.000,E1 138.081} C_DIS
LIN {X 0.095,Y -570.316,Z 1329.567,A 0.000,B 0.000,C 90.000,E1 137.957} C_DIS
LIN {X 0.133,Y -573.302,Z 1329.566,A 0.000,B 0.000,C 90.000,E1 137.838} C_DIS
LIN {X 0.042,Y -579.306,Z 1329.564,A 0.000,B 0.000,C 90.000,E1 137.553} C_DIS
LIN {X 0.041,Y -582.221,Z 1329.563,A 0.000,B 0.000,C 90.000,E1 137.391} C_DIS
LIN {X -0.086,Y -587.902,Z 1329.561,A 0.000,B 0.000,C 90.000,E1 137.025} C_DIS
LIN {X 0.069,Y -593.498,Z 1329.559,A 0.000,B 0.000,C 90.000,E1 136.581} C_DIS
LIN {X -0.154,Y -596.296,Z 1329.558,A 0.000,B 0.000,C 90.000,E1 136.377} C_DIS
LIN {X -0.031,Y -601.360,Z 1329.555,A 0.000,B 0.000,C 90.000,E1 135.891} C_DIS
LIN {X 0.147,Y -607.595,Z 1329.552,A 0.000,B 0.000,C 90.000,E1 135.243} C_DIS
LIN {X 0.013,Y -610.067,Z 1329.550,A 0.000,B 0.000,C 90.000,E1 135.000} C_DIS
LIN {X 0.035,Y -615.533,Z 1329.547,A 0.000,B 0.000,C 90.000,E1 134.352} C_DIS
LIN {X -0.292,Y -619.734,Z 1329.544,A 0.000,B 0.000,C 90.000,E1 133.866} C_DIS
LIN {X -0.057,Y -625.491,Z 1329.539,A 0.000,B 0.000,C 90.000,E1 133.095} C_DIS
LIN {X 0.058,Y -630.086,Z 1329.536,A 0.000,B 0.000,C 90.000,E1 132.447} C_DIS
LIN {X 0.068,Y -637.021,Z 1329.530,A 0.000,B 0.000,C 90.000,E1 131.434} C_DIS
LIN {X -0.154,Y -641.276,Z 1329.527,A 0.000,B 0.000,C 90.000,E1 130.825} C_DIS
LIN {X -0.345,Y -646.197,Z 1329.523,A 0.000,B 0.000,C 90.000,E1 130.092} C_DIS
LIN {X -0.073,Y -650.926,Z 1329.518,A 0.000,B 0.000,C 90.000,E1 129.322} C_DIS
LIN {X 0.091,Y -655.208,Z 1329.515,A 0.000,B 0.000,C 90.000,E1 128.588} C_DIS
LIN {X 0.088,Y -658.147,Z 1329.512,A 0.000,B 0.000,C 90.000,E1 128.096} C_DIS
LIN {X 0.108,Y -660.998,Z 1329.509,A 0.000,B 0.000,C 90.000,E1 127.604} C_DIS
LIN {X 0.068,Y -664.272,Z 1329.506,A 0.000,B 0.000,C 90.000,E1 126.996} C_DIS
LIN {X 0.182,Y -667.364,Z 1329.502,A 0.000,B 0.000,C 90.000,E1 126.377} C_DIS
LIN {X 0.268,Y -669.629,Z 1329.500,A 0.000,B 0.000,C 90.000,E1 125.884} C_DIS
LIN {X -0.048,Y -672.772,Z 1329.495,A 0.000,B 0.000,C 90.000,E1 125.185} C_DIS
LIN {X 0.071,Y -674.731,Z 1329.493,A 0.000,B 0.000,C 90.000,E1 124.692} C_DIS
LIN {X -0.198,Y -677.338,Z 1329.489,A 0.000,B 0.000,C 90.000,E1 123.992} C_DIS
LIN {X 0.120,Y -679.594,Z 1329.485,A 0.000,B 0.000,C 90.000,E1 123.245} C_DIS
LIN {X 0.079,Y -682.147,Z 1329.479,A 0.000,B 0.000,C 90.000,E1 122.291} C_DIS
LIN {X 0.252,Y -683.276,Z 1329.477,A 0.000,B 0.000,C 90.000,E1 121.799} C_DIS
LIN {X -0.312,Y -684.785,Z 1329.473,A 0.000,B 0.000,C 90.000,E1 121.131} C_DIS
LIN {X 0.075,Y -686.136,Z 1329.469,A 0.000,B 0.000,C 90.000,E1 120.384} C_DIS
LIN {X -0.089,Y -686.945,Z 1329.466,A 0.000,B 0.000,C 90.000,E1 119.922} C_DIS
LIN {X -0.025,Y -687.813,Z 1329.462,A 0.000,B 0.000,C 90.000,E1 119.205} C_DIS
LIN {X 0.048,Y -688.393,Z 1329.458,A 0.000,B 0.000,C 90.000,E1 118.487} C_DIS
LIN {X 0.127,Y -688.730,Z 1329.454,A 0.000,B 0.000,C 90.000,E1 117.769} C_DIS
LIN {X 0.126,Y -688.900,Z 1329.449,A 0.000,B 0.000,C 90.000,E1 116.821} C_DIS
LIN {X 0.207,Y -688.729,Z 1329.445,A 0.000,B 0.000,C 90.000,E1 116.104} C_DIS
LIN {X -0.018,Y -688.336,Z 1329.441,A 0.000,B 0.000,C 90.000,E1 115.412} C_DIS
LIN {X 0.213,Y -688.142,Z 1329.440,A 0.000,B 0.000,C 90.000,E1 115.155} C_DIS
LIN {X 0.045,Y -687.389,Z 1329.437,A 0.000,B 0.000,C 90.000,E1 114.695} C_DIS
LIN {X 0.208,Y -686.330,Z 1329.435,A 0.000,B 0.000,C 90.000,E1 114.207} C_DIS
LIN {X -0.196,Y -685.667,Z 1329.433,A 0.000,B 0.000,C 90.000,E1 114.003} C_DIS
LIN {X -0.038,Y -683.469,Z 1329.431,A 0.000,B 0.000,C 90.000,E1 113.515} C_DIS
LIN {X 0.068,Y -682.814,Z 1329.430,A 0.000,B 0.000,C 90.000,E1 113.387} C_DIS
LIN {X 0.172,Y -681.811,Z 1329.429,A 0.000,B 0.000,C 90.000,E1 113.259} C_DIS
LIN {X 0.342,Y -677.054,Z 1329.427,A 0.000,B 0.000,C 90.000,E1 112.770} C_DIS
LIN {X -0.155,Y -675.153,Z 1329.426,A 0.000,B 0.000,C 90.000,E1 112.695} C_DIS
LIN {X 0.252,Y -666.634,Z 1329.424,A 0.000,B 0.000,C 90.000,E1 112.280} C_DIS
LIN {X 0.066,Y -661.066,Z 1329.423,A 0.000,B 0.000,C 90.000,E1 112.153} C_DIS
LIN {X -0.077,Y -656.306,Z 1329.423,A 0.000,B 0.000,C 90.000,E1 112.078} C_DIS
LIN {X -0.150,Y -652.355,Z 1329.422,A 0.000,B 0.000,C 90.000,E1 112.025} C_DIS
LIN {X 0.142,Y -644.224,Z 1329.422,A 0.000,B 0.000,C 90.000,E1 111.897} C_DIS
LIN {X 0.011,Y -641.637,Z 1329.421,A 0.000,B 0.000,C 90.000,E1 111.844} C_DIS
LIN {X -0.025,Y -641.596,Z 1329.421,A 0.000,B 0.000,C 90.000,E1 111.844} C_DIS
LIN {X 0.239,Y -642.547,Z 1329.421,A 0.000,B 0.000,C 90.000,E1 111.663} C_DIS
LIN {X -0.148,Y -648.777,Z 1329.416,A 0.000,B 0.000,C 90.000,E1 110.918} C_DIS
LIN {X -0.264,Y -651.659,Z 1329.414,A 0.000,B 0.000,C 90.000,E1 110.556} C_DIS
LIN {X -0.277,Y -655.770,Z 1329.411,A 0.000,B 0.000,C 90.000,E1 109.939} C_DIS
LIN {X -0.259,Y -659.386,Z 1329.407,A 0.000,B 0.000,C 90.000,E1 109.322} C_DIS
LIN {X 0.194,Y -662.420,Z 1329.404,A 0.000,B 0.000,C 90.000,E1 108.671} C_DIS
LIN {X 0.109,Y -665.633,Z 1329.400,A 0.000,B 0.000,C 90.000,E1 107.946} C_DIS
LIN {X -0.028,Y -669.280,Z 1329.394,A 0.000,B 0.000,C 90.000,E1 106.985} C_DIS
LIN {X 0.015,Y -670.913,Z 1329.392,A 0.000,B 0.000,C 90.000,E1 106.496} C_DIS
LIN {X -0.186,Y -673.018,Z 1329.388,A 0.000,B 0.000,C 90.000,E1 105.788} C_DIS
LIN {X -0.128,Y -674.244,Z 1329.385,A 0.000,B 0.000,C 90.000,E1 105.300} C_DIS
LIN {X -0.297,Y -675.859,Z 1329.381,A 0.000,B 0.000,C 90.000,E1 104.592} C_DIS
LIN {X 0.305,Y -676.364,Z 1329.380,A 0.000,B 0.000,C 90.000,E1 104.300} C_DIS
LIN {X 0.161,Y -677.434,Z 1329.376,A 0.000,B 0.000,C 90.000,E1 103.592} C_DIS
LIN {X 0.070,Y -677.982,Z 1329.373,A 0.000,B 0.000,C 90.000,E1 103.119} C_DIS
LIN {X -0.109,Y -678.396,Z 1329.368,A 0.000,B 0.000,C 90.000,E1 102.175} C_DIS
LIN {X 0.283,Y -678.302,Z 1329.364,A 0.000,B 0.000,C 90.000,E1 101.422} C_DIS
LIN {X 0.192,Y -677.934,Z 1329.361,A 0.000,B 0.000,C 90.000,E1 100.950} C_DIS
LIN {X -0.078,Y -676.973,Z 1329.357,A 0.000,B 0.000,C 90.000,E1 100.254} C_DIS
LIN {X -0.184,Y -676.111,Z 1329.354,A 0.000,B 0.000,C 90.000,E1 99.782} C_DIS
LIN {X 0.255,Y -675.001,Z 1329.352,A 0.000,B 0.000,C 90.000,E1 99.265} C_DIS
LIN {X 0.025,Y -673.459,Z 1329.349,A 0.000,B 0.000,C 90.000,E1 98.803} C_DIS
LIN {X -0.284,Y -670.652,Z 1329.345,A 0.000,B 0.000,C 90.000,E1 98.106} C_DIS
LIN {X 0.129,Y -668.519,Z 1329.342,A 0.000,B 0.000,C 90.000,E1 97.587} C_DIS
LIN {X -0.231,Y -664.930,Z 1329.338,A 0.000,B 0.000,C 90.000,E1 96.891} C_DIS
LIN {X 0.230,Y -663.018,Z 1329.336,A 0.000,B 0.000,C 90.000,E1 96.486} C_DIS
LIN {X -0.171,Y -659.580,Z 1329.333,A 0.000,B 0.000,C 90.000,E1 95.910} C_DIS
LIN {X 0.158,Y -656.571,Z 1329.330,A 0.000,B 0.000,C 90.000,E1 95.391} C_DIS
LIN {X -0.292,Y -652.419,Z 1329.327,A 0.000,B 0.000,C 90.000,E1 94.816} C_DIS
LIN {X -0.173,Y -647.883,Z 1329.323,A 0.000,B 0.000,C 90.000,E1 94.188} C_DIS
LIN {X 0.185,Y -645.051,Z 1329.321,A 0.000,B 0.000,C 90.000,E1 93.784} C_DIS
LIN {X -0.273,Y -640.968,Z 1329.318,A 0.000,B 0.000,C 90.000,E1 93.326} C_DIS
LIN {X -0.080,Y -636.497,Z 1329.316,A 0.000,B 0.000,C 90.000,E1 92.808} C_DIS
LIN {X -0.087,Y -629.111,Z 1329.312,A 0.000,B 0.000,C 90.000,E1 92.064} C_DIS
LIN {X 0.072,Y -622.750,Z 1329.308,A 0.000,B 0.000,C 90.000,E1 91.432} C_DIS
LIN {X -0.257,Y -617.524,Z 1329.305,A 0.000,B 0.000,C 90.000,E1 90.974} C_DIS
LIN {X 0.290,Y -614.711,Z 1329.304,A 0.000,B 0.000,C 90.000,E1 90.688} C_DIS
LIN {X -0.208,Y -609.079,Z 1329.302,A 0.000,B 0.000,C 90.000,E1 90.286} C_DIS
LIN {X -0.142,Y -602.589,Z 1329.299,A 0.000,B 0.000,C 90.000,E1 89.885} C_DIS
LIN {X -0.266,Y -595.681,Z 1329.297,A 0.000,B 0.000,C 90.000,E1 89.542} C_DIS
LIN {X 0.082,Y -588.477,Z 1329.296,A 0.000,B 0.000,C 90.000,E1 89.198} C_DIS
LIN {X 0.167,Y -581.408,Z 1329.294,A 0.000,B 0.000,C 90.000,E1 88.912} C_DIS
LIN {X -0.144,Y -576.842,Z 1329.293,A 0.000,B 0.000,C 90.000,E1 88.740} C_DIS
LIN {X 0.222,Y -574.221,Z 1329.292,A 0.000,B 0.000,C 90.000,E1 88.511} C_DIS
LIN {X 0.230,Y -572.964,Z 1329.291,A 0.000,B 0.000,C 90.000,E1 88.396} C_DIS
LIN {X 0.196,Y -572.941,Z 1329.291,A 0.000,B 0.000,C 90.000,E1 88.396} C_DIS
LIN {X 0.108,Y -572.266,Z 1329.290,A 0.000,B 0.000,C 90.000,E1 88.165} C_DIS
LIN {X -0.107,Y -572.072,Z 1329.289,A 0.000,B 0.000,C 90.000,E1 88.051} C_DIS
LIN {X -0.165,Y -572.033,Z 1329.287,A 0.000,B 0.000,C 90.000,E1 87.650} C_DIS
LIN {X 0.024,Y -574.205,Z 1329.273,A 0.000,B 0.000,C 90.000,E1 85.179} C_DIS
LIN {X 0.129,Y -576.696,Z 1329.261,A 0.000,B 0.000,C 90.000,E1 82.996} C_DIS
LIN {X -0.052,Y -578.331,Z 1329.254,A 0.000,B 0.000,C 90.000,E1 81.659} C_DIS
LIN {X -0.063,Y -580.256,Z 1329.245,A 0.000,B 0.000,C 90.000,E1 80.038} C_DIS
LIN {X 0.275,Y -581.479,Z 1329.239,A 0.000,B 0.000,C 90.000,E1 78.926} C_DIS
LIN {X -0.053,Y -582.617,Z 1329.233,A 0.000,B 0.000,C 90.000,E1 77.881} C_DIS
LIN {X -0.212,Y -583.961,Z 1329.224,A 0.000,B 0.000,C 90.000,E1 76.284} C_DIS
LIN {X 0.173,Y -584.773,Z 1329.218,A 0.000,B 0.000,C 90.000,E1 75.172} C_DIS
LIN {X -0.110,Y -586.092,Z 1329.207,A 0.000,B 0.000,C 90.000,E1 73.323} C_DIS
LIN {X 0.140,Y -587.093,Z 1329.198,A 0.000,B 0.000,C 90.000,E1 71.692} C_DIS
LIN {X -0.007,Y -587.975,Z 1329.191,A 0.000,B 0.000,C 90.000,E1 70.369} C_DIS
LIN {X 0.020,Y -589.382,Z 1329.179,A 0.000,B 0.000,C 90.000,E1 68.230} C_DIS
LIN {X 0.091,Y -590.555,Z 1329.169,A 0.000,B 0.000,C 90.000,E1 66.357} C_DIS
LIN {X -0.244,Y -591.682,Z 1329.160,A 0.000,B 0.000,C 90.000,E1 64.793} C_DIS
LIN {X -0.045,Y -592.859,Z 1329.151,A 0.000,B 0.000,C 90.000,E1 63.179} C_DIS
LIN {X 0.002,Y -594.552,Z 1329.139,A 0.000,B 0.000,C 90.000,E1 61.051} C_DIS
LIN {X -0.058,Y -596.346,Z 1329.129,A 0.000,B 0.000,C 90.000,E1 59.203} C_DIS
LIN {X 0.226,Y -598.230,Z 1329.119,A 0.000,B 0.000,C 90.000,E1 57.327} C_DIS
LIN {X 0.232,Y -599.648,Z 1329.111,A 0.000,B 0.000,C 90.000,E1 56.008} C_DIS
LIN {X 0.267,Y -601.017,Z 1329.104,A 0.000,B 0.000,C 90.000,E1 54.689} C_DIS
LIN {X 0.335,Y -602.722,Z 1329.094,A 0.000,B 0.000,C 90.000,E1 52.844} C_DIS
LIN {X 0.032,Y -603.562,Z 1329.088,A 0.000,B 0.000,C 90.000,E1 51.823} C_DIS
LIN {X -0.212,Y -604.665,Z 1329.079,A 0.000,B 0.000,C 90.000,E1 50.275} C_DIS
LIN {X -0.104,Y -605.260,Z 1329.073,A 0.000,B 0.000,C 90.000,E1 49.218} C_DIS
LIN {X 0.011,Y -605.626,Z 1329.068,A 0.000,B 0.000,C 90.000,E1 48.162} C_DIS
LIN {X -0.129,Y -605.763,Z 1329.063,A 0.000,B 0.000,C 90.000,E1 47.391} C_DIS
LIN {X 0.009,Y -605.987,Z 1329.055,A 0.000,B 0.000,C 90.000,E1 45.810} C_DIS
LIN {X 0.100,Y -605.968,Z 1329.049,A 0.000,B 0.000,C 90.000,E1 44.757} C_DIS
LIN {X 0.381,Y -605.797,Z 1329.044,A 0.000,B 0.000,C 90.000,E1 43.947} C_DIS
LIN {X -0.198,Y -605.554,Z 1329.040,A 0.000,B 0.000,C 90.000,E1 43.218} C_DIS
LIN {X -0.032,Y -605.013,Z 1329.031,A 0.000,B 0.000,C 90.000,E1 41.634} C_DIS
LIN {X -0.119,Y -604.508,Z 1329.024,A 0.000,B 0.000,C 90.000,E1 40.334} C_DIS
LIN {X 0.287,Y -603.552,Z 1329.014,A 0.000,B 0.000,C 90.000,E1 38.463} C_DIS
LIN {X -0.264,Y -603.084,Z 1329.010,A 0.000,B 0.000,C 90.000,E1 37.729} C_DIS
LIN {X -0.342,Y -602.403,Z 1329.005,A 0.000,B 0.000,C 90.000,E1 36.950} C_DIS
LIN {X -0.170,Y -601.048,Z 1328.999,A 0.000,B 0.000,C 90.000,E1 35.884} C_DIS
LIN {X -0.265,Y -599.799,Z 1328.995,A 0.000,B 0.000,C 90.000,E1 35.105} C_DIS
LIN {X -0.139,Y -598.008,Z 1328.989,A 0.000,B 0.000,C 90.000,E1 34.040} C_DIS
LIN {X -0.106,Y -596.365,Z 1328.985,A 0.000,B 0.000,C 90.000,E1 33.245} C_DIS
LIN {X -0.362,Y -593.898,Z 1328.979,A 0.000,B 0.000,C 90.000,E1 32.212} C_DIS
LIN {X -0.254,Y -592.474,Z 1328.976,A 0.000,B 0.000,C 90.000,E1 31.671} C_DIS
LIN {X -0.070,Y -589.141,Z 1328.970,A 0.000,B 0.000,C 90.000,E1 30.590} C_DIS
LIN {X -0.116,Y -586.275,Z 1328.965,A 0.000,B 0.000,C 90.000,E1 29.795} C_DIS
LIN {X -0.193,Y -582.990,Z 1328.961,A 0.000,B 0.000,C 90.000,E1 28.999} C_DIS
LIN {X 0.200,Y -579.337,Z 1328.957,A 0.000,B 0.000,C 90.000,E1 28.153} C_DIS
LIN {X -0.154,Y -575.964,Z 1328.953,A 0.000,B 0.000,C 90.000,E1 27.513} C_DIS
LIN {X -0.021,Y -572.281,Z 1328.949,A 0.000,B 0.000,C 90.000,E1 26.821} C_DIS
LIN {X -0.176,Y -568.254,Z 1328.945,A 0.000,B 0.000,C 90.000,E1 26.155} C_DIS
LIN {X 0.072,Y -565.701,Z 1328.943,A 0.000,B 0.000,C 90.000,E1 25.720} C_DIS
LIN {X 0.115,Y -561.202,Z 1328.939,A 0.000,B 0.000,C 90.000,E1 25.027} C_DIS
LIN {X -0.180,Y -558.267,Z 1328.937,A 0.000,B 0.000,C 90.000,E1 24.643} C_DIS
LIN {X 0.117,Y -551.028,Z 1328.932,A 0.000,B 0.000,C 90.000,E1 23.643} C_DIS
LIN {X 0.030,Y -545.253,Z 1328.928,A 0.000,B 0.000,C 90.000,E1 22.950} C_DIS
LIN {X 0.043,Y -540.685,Z 1328.925,A 0.000,B 0.000,C 90.000,E1 22.408} C_DIS
LIN {X -0.058,Y -533.437,Z 1328.920,A 0.000,B 0.000,C 90.000,E1 21.589} C_DIS
LIN {X -0.210,Y -522.895,Z 1328.914,A 0.000,B 0.000,C 90.000,E1 20.482} C_DIS
LIN {X 0.192,Y -512.268,Z 1328.907,A 0.000,B 0.000,C 90.000,E1 19.322} C_DIS
LIN {X -0.097,Y -503.276,Z 1328.902,A 0.000,B 0.000,C 90.000,E1 18.417} C_DIS
LIN {X 0.051,Y -492.313,Z 1328.896,A 0.000,B 0.000,C 90.000,E1 17.330} C_DIS
LIN {X 0.066,Y -478.032,Z 1328.889,A 0.000,B 0.000,C 90.000,E1 15.969} C_DIS
LIN {X -0.055,Y -470.729,Z 1328.885,A 0.000,B 0.000,C 90.000,E1 15.300} C_DIS
LIN {X 0.171,Y -457.866,Z 1328.878,A 0.000,B 0.000,C 90.000,E1 14.064} C_DIS
LIN {X -0.014,Y -434.965,Z 1328.866,A 0.000,B 0.000,C 90.000,E1 11.827} C_DIS
LIN {X 0.027,Y -419.292,Z 1328.856,A 0.000,B 0.000,C 90.000,E1 10.141} C_DIS
LIN {X -0.049,Y -405.064,Z 1328.848,A 0.000,B 0.000,C 90.000,E1 8.568} C_DIS
LIN {X -0.144,Y -399.403,Z 1328.844,A 0.000,B 0.000,C 90.000,E1 7.936} C_DIS
LIN {X 0.014,Y -395.330,Z 1328.841,A 0.000,B 0.000,C 90.000,E1 7.352} C_DIS
LIN {X -0.021,Y -395.342,Z 1328.841,A 0.000,B 0.000,C 90.000,E1 7.352} C_DIS
LIN {X 0.173,Y -395.735,Z 1328.840,A 0.000,B 0.000,C 90.000,E1 7.182} C_DIS
LIN {X 0.135,Y -395.790,Z 1328.840,A 0.000,B 0.000,C 90.000,E1 7.182} C_DIS
LIN {X 0.064,Y -399.630,Z 1328.838,A 0.000,B 0.000,C 90.000,E1 6.834} C_DIS
LIN {X -0.003,Y -413.923,Z 1328.833,A 0.000,B 0.000,C 90.000,E1 5.910} C_DIS
LIN {X 0.077,Y -417.183,Z 1328.832,A 0.000,B 0.000,C 90.000,E1 5.682} C_DIS
LIN {X 0.049,Y -423.391,Z 1328.829,A 0.000,B 0.000,C 90.000,E1 5.220} C_DIS
LIN {X 0.201,Y -429.465,Z 1328.826,A 0.000,B 0.000,C 90.000,E1 4.702} C_DIS
LIN {X -0.119,Y -436.877,Z 1328.823,A 0.000,B 0.000,C 90.000,E1 4.073} C_DIS
LIN {X 0.013,Y -442.747,Z 1328.819,A 0.000,B 0.000,C 90.000,E1 3.498} C_DIS
LIN {X -0.014,Y -448.465,Z 1328.816,A 0.000,B 0.000,C 90.000,E1 2.922} C_DIS
LIN {X -0.159,Y -454.063,Z 1328.813,A 0.000,B 0.000,C 90.000,E1 2.350} C_DIS
LIN {X 0.134,Y -460.792,Z 1328.809,A 0.000,B 0.000,C 90.000,E1 1.547} C_DIS
LIN {X -0.220,Y -467.202,Z 1328.804,A 0.000,B 0.000,C 90.000,E1 0.802} C_DIS
LIN {X -0.174,Y -471.978,Z 1328.801,A 0.000,B 0.000,C 90.000,E1 0.172} C_DIS
LIN {X 0.097,Y -477.741,Z 1328.796,A 0.000,B 0.000,C 90.000,E1 359.312} C_DIS
LIN {X -0.163,Y -482.716,Z 1328.792,A 0.000,B 0.000,C 90.000,E1 358.568} C_DIS
LIN {X -0.050,Y -489.012,Z 1328.786,A 0.000,B 0.000,C 90.000,E1 357.478} C_DIS
LIN {X -0.056,Y -491.585,Z 1328.783,A 0.000,B 0.000,C 90.000,E1 357.020} C_DIS
LIN {X -0.171,Y -495.517,Z 1328.779,A 0.000,B 0.000,C 90.000,E1 356.274} C_DIS
LIN {X -0.251,Y -499.138,Z 1328.775,A 0.000,B 0.000,C 90.000,E1 355.527} C_DIS
LIN {X 0.204,Y -502.536,Z 1328.771,A 0.000,B 0.000,C 90.000,E1 354.723} C_DIS
LIN {X -0.001,Y -505.083,Z 1328.768,A 0.000,B 0.000,C 90.000,E1 354.147} C_DIS
LIN {X 0.063,Y -508.027,Z 1328.763,A 0.000,B 0.000,C 90.000,E1 353.394} C_DIS
LIN {X -0.152,Y -511.392,Z 1328.758,A 0.000,B 0.000,C 90.000,E1 352.527} C_DIS
LIN {X 0.177,Y -514.367,Z 1328.754,A 0.000,B 0.000,C 90.000,E1 351.602} C_DIS
LIN {X 0.009,Y -517.780,Z 1328.747,A 0.000,B 0.000,C 90.000,E1 350.443} C_DIS
LIN {X -0.019,Y -520.165,Z 1328.742,A 0.000,B 0.000,C 90.000,E1 349.567} C_DIS
LIN {X -0.119,Y -522.204,Z 1328.737,A 0.000,B 0.000,C 90.000,E1 348.701} C_DIS
LIN {X 0.008,Y -524.037,Z 1328.732,A 0.000,B 0.000,C 90.000,E1 347.813} C_DIS
LIN {X 0.067,Y -526.138,Z 1328.726,A 0.000,B 0.000,C 90.000,E1 346.645} C_DIS
LIN {X 0.102,Y -527.057,Z 1328.723,A 0.000,B 0.000,C 90.000,E1 346.061} C_DIS
LIN {X -0.195,Y -528.532,Z 1328.716,A 0.000,B 0.000,C 90.000,E1 344.936} C_DIS
LIN {X 0.158,Y -529.427,Z 1328.711,A 0.000,B 0.000,C 90.000,E1 344.031} C_DIS
LIN {X -0.129,Y -530.038,Z 1328.707,A 0.000,B 0.000,C 90.000,E1 343.196} C_DIS
LIN {X 0.071,Y -530.303,Z 1328.703,A 0.000,B 0.000,C 90.000,E1 342.598} C_DIS
LIN {X -0.029,Y -530.458,Z 1328.697,A 0.000,B 0.000,C 90.000,E1 341.456} C_DIS
LIN {X -0.144,Y -530.299,Z 1328.692,A 0.000,B 0.000,C 90.000,E1 340.604} C_DIS
LIN {X -0.074,Y -529.454,Z 1328.686,A 0.000,B 0.000,C 90.000,E1 339.444} C_DIS
LIN {X 0.108,Y -528.895,Z 1328.683,A 0.000,B 0.000,C 90.000,E1 338.847} C_DIS
LIN {X -0.018,Y -528.069,Z 1328.679,A 0.000,B 0.000,C 90.000,E1 338.284} C_DIS
LIN {X -0.102,Y -525.579,Z 1328.671,A 0.000,B 0.000,C 90.000,E1 336.847} C_DIS
LIN {X -0.075,Y -523.747,Z 1328.667,A 0.000,B 0.000,C 90.000,E1 335.973} C_DIS
LIN {X -0.072,Y -521.541,Z 1328.662,A 0.000,B 0.000,C 90.000,E1 335.101} C_DIS
LIN {X 0.265,Y -517.981,Z 1328.655,A 0.000,B 0.000,C 90.000,E1 333.896} C_DIS
LIN {X -0.258,Y -513.402,Z 1328.647,A 0.000,B 0.000,C 90.000,E1 332.487} C_DIS
LIN {X 0.072,Y -508.673,Z 1328.639,A 0.000,B 0.000,C 90.000,E1 330.973} C_DIS
LIN {X 0.043,Y -506.628,Z 1328.635,A 0.000,B 0.000,C 90.000,E1 330.383} C_DIS
LIN {X -0.002,Y -504.241,Z 1328.632,A 0.000,B 0.000,C 90.000,E1 329.793} C_DIS
LIN {X 0.120,Y -502.186,Z 1328.630,A 0.000,B 0.000,C 90.000,E1 329.331} C_DIS
LIN {X 0.230,Y -499.534,Z 1328.627,A 0.000,B 0.000,C 90.000,E1 328.869} C_DIS
LIN {X -0.162,Y -497.324,Z 1328.626,A 0.000,B 0.000,C 90.000,E1 328.614} C_DIS
LIN {X -0.102,Y -495.892,Z 1328.625,A 0.000,B 0.000,C 90.000,E1 328.456} C_DIS
LIN {X -0.150,Y -466.078,Z 1328.612,A 0.000,B 0.000,C 90.000,E1 326.215} C_DIS
LIN {X -0.092,Y -443.582,Z 1328.602,A 0.000,B 0.000,C 90.000,E1 324.276} C_DIS
LIN {X 0.083,Y -423.107,Z 1328.590,A 0.000,B 0.000,C 90.000,E1 322.271} C_DIS
LIN {X -0.044,Y -404.612,Z 1328.579,A 0.000,B 0.000,C 90.000,E1 320.275} C_DIS
LIN {X -0.078,Y -386.671,Z 1328.567,A 0.000,B 0.000,C 90.000,E1 318.081} C_DIS
LIN {X -0.101,Y -378.491,Z 1328.561,A 0.000,B 0.000,C 90.000,E1 316.986} C_DIS
LIN {X -0.138,Y -378.460,Z 1328.561,A 0.000,B 0.000,C 90.000,E1 316.986} C_DIS
LIN {X -0.067,Y -384.122,Z 1328.530,A 0.000,B 0.000,C 90.000,E1 311.391} C_DIS
LIN {X -0.024,Y -384.622,Z 1328.528,A 0.000,B 0.000,C 90.000,E1 311.024} C_DIS
LIN {X 0.029,Y -385.224,Z 1328.524,A 0.000,B 0.000,C 90.000,E1 310.297} C_DIS
LIN {X 0.067,Y -391.278,Z 1328.492,A 0.000,B 0.000,C 90.000,E1 304.565} C_DIS
LIN {X -0.102,Y -396.991,Z 1328.459,A 0.000,B 0.000,C 90.000,E1 298.565} C_DIS
LIN {X -0.151,Y -401.356,Z 1328.427,A 0.000,B 0.000,C 90.000,E1 292.950} C_DIS
LIN {X -0.071,Y -401.658,Z 1328.426,A 0.000,B 0.000,C 90.000,E1 292.589} C_DIS
LIN {X 0.081,Y -404.750,Z 1328.395,A 0.000,B 0.000,C 90.000,E1 286.985} C_DIS
LIN {X 0.095,Y -406.157,Z 1328.364,A 0.000,B 0.000,C 90.000,E1 281.422} C_DIS
LIN {X 0.199,Y -405.674,Z 1328.333,A 0.000,B 0.000,C 90.000,E1 275.853} C_DIS
LIN {X -0.133,Y -403.564,Z 1328.306,A 0.000,B 0.000,C 90.000,E1 271.031} C_DIS
LIN {X -0.198,Y -403.167,Z 1328.302,A 0.000,B 0.000,C 90.000,E1 270.344} C_DIS
LIN {X 0.035,Y -399.061,Z 1328.273,A 0.000,B 0.000,C 90.000,E1 265.065} C_DIS
LIN {X -0.023,Y -398.758,Z 1328.271,A 0.000,B 0.000,C 90.000,E1 264.723} C_DIS
LIN {X -0.133,Y -393.282,Z 1328.243,A 0.000,B 0.000,C 90.000,E1 259.803} C_DIS
LIN {X 0.174,Y -392.650,Z 1328.239,A 0.000,B 0.000,C 90.000,E1 259.050} C_DIS
LIN {X -0.040,Y -386.234,Z 1328.214,A 0.000,B 0.000,C 90.000,E1 254.448} C_DIS
LIN {X -0.075,Y -385.136,Z 1328.208,A 0.000,B 0.000,C 90.000,E1 253.378} C_DIS
LIN {X 0.034,Y -377.799,Z 1328.182,A 0.000,B 0.000,C 90.000,E1 248.666} C_DIS
LIN {X -0.095,Y -376.066,Z 1328.173,A 0.000,B 0.000,C 90.000,E1 247.230} C_DIS
LIN {X -0.037,Y -368.735,Z 1328.149,A 0.000,B 0.000,C 90.000,E1 242.820} C_DIS
LIN {X -0.052,Y -366.383,Z 1328.139,A 0.000,B 0.000,C 90.000,E1 240.973} C_DIS
LIN {X 0.114,Y -365.078,Z 1328.135,A 0.000,B 0.000,C 90.000,E1 240.205} C_DIS
LIN {X 0.161,Y -358.486,Z 1328.112,A 0.000,B 0.000,C 90.000,E1 236.087} C_DIS
LIN {X 0.212,Y -356.164,Z 1328.101,A 0.000,B 0.000,C 90.000,E1 234.196} C_DIS
LIN {X -0.137,Y -354.910,Z 1328.097,A 0.000,B 0.000,C 90.000,E1 233.497} C_DIS
LIN {X -0.153,Y -348.144,Z 1328.072,A 0.000,B 0.000,C 90.000,E1 228.933} C_DIS
LIN {X 0.182,Y -347.402,Z 1328.068,A 0.000,B 0.000,C 90.000,E1 228.243} C_DIS
LIN {X 0.164,Y -347.418,Z 1328.068,A 0.000,B 0.000,C 90.000,E1 228.243} C_DIS
LIN {X -0.202,Y -361.731,Z 1328.055,A 0.000,B 0.000,C 90.000,E1 225.891} C_DIS
LIN {X -0.065,Y -377.937,Z 1328.042,A 0.000,B 0.000,C 90.000,E1 223.461} C_DIS
LIN {X -0.180,Y -395.714,Z 1328.029,A 0.000,B 0.000,C 90.000,E1 221.148} C_DIS
LIN {X -0.137,Y -414.284,Z 1328.017,A 0.000,B 0.000,C 90.000,E1 218.991} C_DIS
LIN {X -0.074,Y -434.892,Z 1328.005,A 0.000,B 0.000,C 90.000,E1 216.870} C_DIS
LIN {X -0.141,Y -442.392,Z 1328.001,A 0.000,B 0.000,C 90.000,E1 216.171} C_DIS
LIN {X -0.061,Y -444.621,Z 1327.999,A 0.000,B 0.000,C 90.000,E1 215.884} C_DIS
LIN {X 0.241,Y -446.074,Z 1327.998,A 0.000,B 0.000,C 90.000,E1 215.518} C_DIS
LIN {X -0.067,Y -447.124,Z 1327.996,A 0.000,B 0.000,C 90.000,E1 215.231} C_DIS
LIN {X 0.060,Y -448.708,Z 1327.992,A 0.000,B 0.000,C 90.000,E1 214.565} C_DIS
LIN {X 0.085,Y -449.900,Z 1327.989,A 0.000,B 0.000,C 90.000,E1 213.913} C_DIS
LIN {X -0.052,Y -451.299,Z 1327.983,A 0.000,B 0.000,C 90.000,E1 212.959} C_DIS
LIN {X 0.010,Y -453.039,Z 1327.974,A 0.000,B 0.000,C 90.000,E1 211.337} C_DIS
LIN {X -0.026,Y -455.177,Z 1327.963,A 0.000,B 0.000,C 90.000,E1 209.411} C_DIS
LIN {X -0.131,Y -458.838,Z 1327.947,A 0.000,B 0.000,C 90.000,E1 206.539} C_DIS
LIN {X 0.069,Y -462.151,Z 1327.935,A 0.000,B 0.000,C 90.000,E1 204.283} C_DIS
LIN {X 0.004,Y -464.724,Z 1327.924,A 0.000,B 0.000,C 90.000,E1 202.386} C_DIS
LIN {X 0.122,Y -466.834,Z 1327.916,A 0.000,B 0.000,C 90.000,E1 200.791} C_DIS
LIN {X 0.122,Y -468.858,Z 1327.907,A 0.000,B 0.000,C 90.000,E1 199.214} C_DIS
LIN {X -0.234,Y -470.444,Z 1327.900,A 0.000,B 0.000,C 90.000,E1 198.000} C_DIS
LIN {X 0.143,Y -472.483,Z 1327.891,A 0.000,B 0.000,C 90.000,E1 196.386} C_DIS
LIN {X -0.069,Y -474.699,Z 1327.881,A 0.000,B 0.000,C 90.000,E1 194.537} C_DIS
LIN {X 0.100,Y -476.930,Z 1327.870,A 0.000,B 0.000,C 90.000,E1 192.647} C_DIS
LIN {X 0.117,Y -479.192,Z 1327.860,A 0.000,B 0.000,C 90.000,E1 190.782} C_DIS
LIN {X -0.141,Y -481.012,Z 1327.851,A 0.000,B 0.000,C 90.000,E1 189.265} C_DIS
LIN {X 0.169,Y -482.465,Z 1327.845,A 0.000,B 0.000,C 90.000,E1 187.992} C_DIS
LIN {X -0.118,Y -484.032,Z 1327.836,A 0.000,B 0.000,C 90.000,E1 186.486} C_DIS
LIN {X 0.180,Y -485.159,Z 1327.829,A 0.000,B 0.000,C 90.000,E1 185.220} C_DIS
LIN {X 0.012,Y -486.201,Z 1327.822,A 0.000,B 0.000,C 90.000,E1 184.012} C_DIS
LIN {X 0.144,Y -486.642,Z 1327.819,A 0.000,B 0.000,C 90.000,E1 183.383} C_DIS
LIN {X -0.199,Y -487.421,Z 1327.810,A 0.000,B 0.000,C 90.000,E1 181.892} C_DIS
LIN {X -0.201,Y -487.760,Z 1327.805,A 0.000,B 0.000,C 90.000,E1 180.974} C_DIS
LIN {X -0.210,Y -487.959,Z 1327.800,A 0.000,B 0.000,C 90.000,E1 180.057} C_DIS
LIN {X 0.106,Y -488.039,Z 1327.793,A 0.000,B 0.000,C 90.000,E1 178.797} C_DIS
LIN {X 0.111,Y -487.871,Z 1327.788,A 0.000,B 0.000,C 90.000,E1 177.879} C_DIS
LIN {X 0.095,Y -487.542,Z 1327.783,A 0.000,B 0.000,C 90.000,E1 176.963} C_DIS
LIN {X -0.042,Y -486.721,Z 1327.776,A 0.000,B 0.000,C 90.000,E1 175.755} C_DIS
LIN {X -0.048,Y -485.882,Z 1327.771,A 0.000,B 0.000,C 90.000,E1 174.837} C_DIS
LIN {X -0.207,Y -484.377,Z 1327.765,A 0.000,B 0.000,C 90.000,E1 173.628} C_DIS
LIN {X -0.195,Y -482.912,Z 1327.759,A 0.000,B 0.000,C 90.000,E1 172.704} C_DIS
LIN {X 0.008,Y -481.759,Z 1327.756,A 0.000,B 0.000,C 90.000,E1 172.064} C_DIS
LIN {X -0.008,Y -479.736,Z 1327.751,A 0.000,B 0.000,C 90.000,E1 171.141} C_DIS
LIN {X 0.028,Y -477.116,Z 1327.746,A 0.000,B 0.000,C 90.000,E1 170.208} C_DIS
LIN {X 0.106,Y -475.212,Z 1327.742,A 0.000,B 0.000,C 90.000,E1 169.577} C_DIS
LIN {X 0.144,Y -473.334,Z 1327.740,A 0.000,B 0.000,C 90.000,E1 169.106} C_DIS
LIN {X 0.003,Y -469.796,Z 1327.735,A 0.000,B 0.000,C 90.000,E1 168.342} C_DIS
LIN {X -0.087,Y -464.212,Z 1327.730,A 0.000,B 0.000,C 90.000,E1 167.409} C_DIS
LIN {X -0.026,Y -454.213,Z 1327.721,A 0.000,B 0.000,C 90.000,E1 165.811} C_DIS
LIN {X -0.014,Y -443.021,Z 1327.711,A 0.000,B 0.000,C 90.000,E1 164.031} C_DIS
LIN {X 0.111,Y -438.107,Z 1327.707,A 0.000,B 0.000,C 90.000,E1 163.196} C_DIS
LIN {X 0.064,Y -434.591,Z 1327.703,A 0.000,B 0.000,C 90.000,E1 162.543} C_DIS
LIN {X -0.113,Y -433.185,Z 1327.701,A 0.000,B 0.000,C 90.000,E1 162.236} C_DIS
LIN {X 0.120,Y -431.995,Z 1327.699,A 0.000,B 0.000,C 90.000,E1 161.873} C_DIS
LIN {X -0.198,Y -431.251,Z 1327.698,A 0.000,B 0.000,C 90.000,E1 161.583} C_DIS
LIN {X 0.117,Y -430.804,Z 1327.695,A 0.000,B 0.000,C 90.000,E1 161.094} C_DIS
LIN {X 0.079,Y -430.821,Z 1327.695,A 0.000,B 0.000,C 90.000,E1 161.094} C_DIS
LIN {X -0.164,Y -431.634,Z 1327.694,A 0.000,B 0.000,C 90.000,E1 160.913} C_DIS
LIN {X -0.118,Y -432.284,Z 1327.693,A 0.000,B 0.000,C 90.000,E1 160.678} C_DIS
LIN {X -0.158,Y -432.313,Z 1327.693,A 0.000,B 0.000,C 90.000,E1 160.678} C_DIS
LIN {X -0.175,Y -434.643,Z 1327.691,A 0.000,B 0.000,C 90.000,E1 160.423} C_DIS
LIN {X 0.176,Y -440.078,Z 1327.688,A 0.000,B 0.000,C 90.000,E1 159.880} C_DIS
LIN {X 0.105,Y -441.563,Z 1327.688,A 0.000,B 0.000,C 90.000,E1 159.752} C_DIS
LIN {X 0.140,Y -459.463,Z 1327.680,A 0.000,B 0.000,C 90.000,E1 158.337} C_DIS
LIN {X 0.050,Y -473.230,Z 1327.674,A 0.000,B 0.000,C 90.000,E1 157.283} C_DIS
LIN {X 0.163,Y -482.174,Z 1327.670,A 0.000,B 0.000,C 90.000,E1 156.538} C_DIS
LIN {X -0.036,Y -487.973,Z 1327.667,A 0.000,B 0.000,C 90.000,E1 156.049} C_DIS
LIN {X 0.108,Y -496.565,Z 1327.662,A 0.000,B 0.000,C 90.000,E1 155.229} C_DIS
LIN {X 0.146,Y -503.321,Z 1327.659,A 0.000,B 0.000,C 90.000,E1 154.537} C_DIS
LIN {X -0.266,Y -508.621,Z 1327.656,A 0.000,B 0.000,C 90.000,E1 154.024} C_DIS
LIN {X -0.147,Y -513.759,Z 1327.652,A 0.000,B 0.000,C 90.000,E1 153.435} C_DIS
LIN {X -0.210,Y -517.488,Z 1327.650,A 0.000,B 0.000,C 90.000,E1 152.999} C_DIS
LIN {X -0.019,Y -521.020,Z 1327.647,A 0.000,B 0.000,C 90.000,E1 152.538} C_DIS
LIN {X -0.209,Y -525.158,Z 1327.644,A 0.000,B 0.000,C 90.000,E1 151.975} C_DIS
LIN {X -0.124,Y -528.777,Z 1327.641,A 0.000,B 0.000,C 90.000,E1 151.385} C_DIS
LIN {X -0.161,Y -532.500,Z 1327.637,A 0.000,B 0.000,C 90.000,E1 150.667} C_DIS
LIN {X 0.101,Y -535.429,Z 1327.633,A 0.000,B 0.000,C 90.000,E1 149.921} C_DIS
LIN {X 0.263,Y -537.337,Z 1327.630,A 0.000,B 0.000,C 90.000,E1 149.331} C_DIS
LIN {X -0.306,Y -539.784,Z 1327.625,A 0.000,B 0.000,C 90.000,E1 148.535} C_DIS
LIN {X -0.108,Y -541.852,Z 1327.620,A 0.000,B 0.000,C 90.000,E1 147.661} C_DIS
LIN {X -0.072,Y -543.032,Z 1327.617,A 0.000,B 0.000,C 90.000,E1 147.089} C_DIS
LIN {X 0.164,Y -544.535,Z 1327.612,A 0.000,B 0.000,C 90.000,E1 146.215} C_DIS
LIN {X -0.043,Y -545.758,Z 1327.608,A 0.000,B 0.000,C 90.000,E1 145.388} C_DIS
LIN {X -0.198,Y -547.012,Z 1327.601,A 0.000,B 0.000,C 90.000,E1 144.276} C_DIS
LIN {X -0.064,Y -547.737,Z 1327.597,A 0.000,B 0.000,C 90.000,E1 143.417} C_DIS
LIN {X 0.177,Y -548.698,Z 1327.589,A 0.000,B 0.000,C 90.000,E1 141.984} C_DIS
LIN {X 0.048,Y -549.947,Z 1327.580,A 0.000,B 0.000,C 90.000,E1 140.312} C_DIS
LIN {X 0.082,Y -550.567,Z 1327.576,A 0.000,B 0.000,C 90.000,E1 139.747} C_DIS
LIN {X 0.102,Y -551.179,Z 1327.575,A 0.000,B 0.000,C 90.000,E1 139.461} C_DIS
LIN {X 0.059,Y -551.218,Z 1327.575,A 0.000,B 0.000,C 90.000,E1 139.461} C_DIS
LIN {X 0.181,Y -552.459,Z 1327.574,A 0.000,B 0.000,C 90.000,E1 139.299} C_DIS
LIN {X 0.132,Y -553.662,Z 1327.573,A 0.000,B 0.000,C 90.000,E1 139.094} C_DIS
LIN {X 0.278,Y -553.910,Z 1327.573,A 0.000,B 0.000,C 90.000,E1 139.013} C_DIS
LIN {X 0.236,Y -553.951,Z 1327.573,A 0.000,B 0.000,C 90.000,E1 139.013} C_DIS
LIN {X -0.120,Y -557.358,Z 1327.571,A 0.000,B 0.000,C 90.000,E1 138.852} C_DIS
LIN {X 0.116,Y -564.294,Z 1327.570,A 0.000,B 0.000,C 90.000,E1 138.647} C_DIS
LIN {X 0.102,Y -570.646,Z 1327.569,A 0.000,B 0.000,C 90.000,E1 138.447} C_DIS
LIN {X 0.357,Y -576.542,Z 1327.568,A 0.000,B 0.000,C 90.000,E1 138.162} C_DIS
LIN {X -0.085,Y -582.258,Z 1327.566,A 0.000,B 0.000,C 90.000,E1 137.877} C_DIS
LIN {X 0.041,Y -588.071,Z 1327.564,A 0.000,B 0.000,C 90.000,E1 137.472} C_DIS
LIN {X -0.190,Y -593.631,Z 1327.561,A 0.000,B 0.000,C 90.000,E1 137.067} C_DIS
LIN {X 0.097,Y -598.881,Z 1327.559,A 0.000,B 0.000,C 90.000,E1 136.581} C_DIS
LIN {X -0.381,Y -603.844,Z 1327.556,A 0.000,B 0.000,C 90.000,E1 136.134} C_DIS
LIN {X 0.268,Y -608.614,Z 1327.553,A 0.000,B 0.000,C 90.000,E1 135.567} C_DIS
LIN {X 0.081,Y -611.052,Z 1327.552,A 0.000,B 0.000,C 90.000,E1 135.324} C_DIS
LIN {X 0.115,Y -616.427,Z 1327.548,A 0.000,B 0.000,C 90.000,E1 134.676} C_DIS
LIN {X -0.205,Y -620.483,Z 1327.545,A 0.000,B 0.000,C 90.000,E1 134.190} C_DIS
LIN {X 0.278,Y -628.779,Z 1327.539,A 0.000,B 0.000,C 90.000,E1 133.014} C_DIS
LIN {X 0.014,Y -633.991,Z 1327.535,A 0.000,B 0.000,C 90.000,E1 132.285} C_DIS
LIN {X -0.359,Y -642.211,Z 1327.528,A 0.000,B 0.000,C 90.000,E1 131.067} C_DIS
LIN {X -0.123,Y -647.027,Z 1327.524,A 0.000,B 0.000,C 90.000,E1 130.297} C_DIS
LIN {X -0.190,Y -650.152,Z 1327.521,A 0.000,B 0.000,C 90.000,E1 129.806} C_DIS
LIN {X -0.345,Y -656.104,Z 1327.516,A 0.000,B 0.000,C 90.000,E1 128.830} C_DIS
LIN {X 0.098,Y -659.575,Z 1327.512,A 0.000,B 0.000,C 90.000,E1 128.177} C_DIS
LIN {X 0.048,Y -662.916,Z 1327.509,A 0.000,B 0.000,C 90.000,E1 127.569} C_DIS
LIN {X 0.118,Y -665.456,Z 1327.506,A 0.000,B 0.000,C 90.000,E1 127.076} C_DIS
LIN {X 0.184,Y -667.882,Z 1327.503,A 0.000,B 0.000,C 90.000,E1 126.583} C_DIS
LIN {X 0.272,Y -670.085,Z 1327.501,A 0.000,B 0.000,C 90.000,E1 126.091} C_DIS
LIN {X -0.041,Y -673.180,Z 1327.497,A 0.000,B 0.000,C 90.000,E1 125.391} C_DIS
LIN {X 0.060,Y -675.970,Z 1327.493,A 0.000,B 0.000,C 90.000,E1 124.659} C_DIS
LIN {X 0.358,Y -678.431,Z 1327.489,A 0.000,B 0.000,C 90.000,E1 123.913} C_DIS
LIN {X 0.298,Y -681.235,Z 1327.483,A 0.000,B 0.000,C 90.000,E1 122.959} C_DIS
LIN {X 0.276,Y -683.664,Z 1327.478,A 0.000,B 0.000,C 90.000,E1 122.005} C_DIS
LIN {X -0.076,Y -685.632,Z 1327.473,A 0.000,B 0.000,C 90.000,E1 121.082} C_DIS
LIN {X -0.051,Y -687.367,Z 1327.467,A 0.000,B 0.000,C 90.000,E1 120.129} C_DIS
LIN {X 0.018,Y -688.325,Z 1327.464,A 0.000,B 0.000,C 90.000,E1 119.411} C_DIS
LIN {X 0.099,Y -688.974,Z 1327.459,A 0.000,B 0.000,C 90.000,E1 118.693} C_DIS
LIN {X 0.187,Y -689.380,Z 1327.456,A 0.000,B 0.000,C 90.000,E1 117.975} C_DIS
LIN {X -0.104,Y -689.615,Z 1327.450,A 0.000,B 0.000,C 90.000,E1 117.052} C_DIS
LIN {X -0.328,Y -689.552,Z 1327.446,A 0.000,B 0.000,C 90.000,E1 116.360} C_DIS
LIN {X 0.374,Y -689.229,Z 1327.442,A 0.000,B 0.000,C 90.000,E1 115.591} C_DIS
LIN {X -0.079,Y -688.864,Z 1327.440,A 0.000,B 0.000,C 90.000,E1 115.155} C_DIS
LIN {X 0.383,Y -688.108,Z 1327.437,A 0.000,B 0.000,C 90.000,E1 114.643} C_DIS
LIN {X -0.072,Y -687.034,Z 1327.434,A 0.000,B 0.000,C 90.000,E1 114.207} C_DIS
LIN {X 0.152,Y -686.344,Z 1327.433,A 0.000,B 0.000,C 90.000,E1 113.951} C_DIS
LIN {X -0.312,Y -684.106,Z 1327.431,A 0.000,B 0.000,C 90.000,E1 113.515} C_DIS
LIN {X -0.205,Y -683.451,Z 1327.430,A 0.000,B 0.000,C 90.000,E1 113.387} C_DIS
LIN {X -0.098,Y -682.451,Z 1327.429,A 0.000,B 0.000,C 90.000,E1 113.259} C_DIS
LIN {X 0.076,Y -677.625,Z 1327.427,A 0.000,B 0.000,C 90.000,E1 112.770} C_DIS
LIN {X 0.215,Y -675.750,Z 1327.426,A 0.000,B 0.000,C 90.000,E1 112.642} C_DIS
LIN {X -0.050,Y -668.230,Z 1327.424,A 0.000,B 0.000,C 90.000,E1 112.333} C_DIS
LIN {X -0.269,Y -666.200,Z 1327.424,A 0.000,B 0.000,C 90.000,E1 112.280} C_DIS
LIN {X -0.102,Y -663.813,Z 1327.423,A 0.000,B 0.000,C 90.000,E1 112.206} C_DIS
LIN {X -0.175,Y -657.186,Z 1327.423,A 0.000,B 0.000,C 90.000,E1 112.078} C_DIS
LIN {X 0.050,Y -644.146,Z 1327.422,A 0.000,B 0.000,C 90.000,E1 111.897} C_DIS
LIN {X -0.006,Y -641.984,Z 1327.421,A 0.000,B 0.000,C 90.000,E1 111.844} C_DIS
LIN {X -0.071,Y -641.853,Z 1327.421,A 0.000,B 0.000,C 90.000,E1 111.844} C_DIS
LIN {X 0.234,Y -642.665,Z 1327.421,A 0.000,B 0.000,C 90.000,E1 111.663} C_DIS
LIN {X -0.147,Y -648.915,Z 1327.416,A 0.000,B 0.000,C 90.000,E1 110.918} C_DIS
LIN {X -0.262,Y -651.797,Z 1327.414,A 0.000,B 0.000,C 90.000,E1 110.556} C_DIS
LIN {X -0.273,Y -655.872,Z 1327.411,A 0.000,B 0.000,C 90.000,E1 109.939} C_DIS
LIN {X -0.255,Y -659.511,Z 1327.407,A 0.000,B 0.000,C 90.000,E1 109.322} C_DIS
LIN {X 0.199,Y -662.545,Z 1327.404,A 0.000,B 0.000,C 90.000,E1 108.671} C_DIS
LIN {X 0.115,Y -665.763,Z 1327.400,A 0.000,B 0.000,C 90.000,E1 107.946} C_DIS
LIN {X -0.021,Y -669.413,Z 1327.394,A 0.000,B 0.000,C 90.000,E1 106.985} C_DIS
LIN {X 0.024,Y -671.049,Z 1327.392,A 0.000,B 0.000,C 90.000,E1 106.496} C_DIS
LIN {X -0.176,Y -673.156,Z 1327.388,A 0.000,B 0.000,C 90.000,E1 105.788} C_DIS
LIN {X -0.117,Y -674.385,Z 1327.385,A 0.000,B 0.000,C 90.000,E1 105.300} C_DIS
LIN {X -0.284,Y -675.973,Z 1327.381,A 0.000,B 0.000,C 90.000,E1 104.592} C_DIS
LIN {X 0.270,Y -676.852,Z 1327.378,A 0.000,B 0.000,C 90.000,E1 104.064} C_DIS
LIN {X 0.129,Y -677.828,Z 1327.374,A 0.000,B 0.000,C 90.000,E1 103.355} C_DIS
LIN {X 0.085,Y -678.102,Z 1327.373,A 0.000,B 0.000,C 90.000,E1 103.119} C_DIS
LIN {X -0.093,Y -678.547,Z 1327.368,A 0.000,B 0.000,C 90.000,E1 102.175} C_DIS
LIN {X -0.320,Y -678.517,Z 1327.365,A 0.000,B 0.000,C 90.000,E1 101.715} C_DIS
LIN {X 0.257,Y -678.291,Z 1327.362,A 0.000,B 0.000,C 90.000,E1 101.186} C_DIS
LIN {X 0.164,Y -677.835,Z 1327.360,A 0.000,B 0.000,C 90.000,E1 100.715} C_DIS
LIN {X -0.108,Y -676.743,Z 1327.356,A 0.000,B 0.000,C 90.000,E1 100.018} C_DIS
LIN {X -0.331,Y -675.771,Z 1327.353,A 0.000,B 0.000,C 90.000,E1 99.557} C_DIS
LIN {X 0.279,Y -675.229,Z 1327.352,A 0.000,B 0.000,C 90.000,E1 99.265} C_DIS
LIN {X 0.050,Y -673.690,Z 1327.349,A 0.000,B 0.000,C 90.000,E1 98.803} C_DIS
LIN {X -0.257,Y -670.890,Z 1327.345,A 0.000,B 0.000,C 90.000,E1 98.106} C_DIS
LIN {X 0.156,Y -668.758,Z 1327.342,A 0.000,B 0.000,C 90.000,E1 97.587} C_DIS
LIN {X -0.201,Y -665.171,Z 1327.338,A 0.000,B 0.000,C 90.000,E1 96.891} C_DIS
LIN {X 0.261,Y -663.263,Z 1327.336,A 0.000,B 0.000,C 90.000,E1 96.486} C_DIS
LIN {X -0.228,Y -659.031,Z 1327.332,A 0.000,B 0.000,C 90.000,E1 95.796} C_DIS
LIN {X 0.199,Y -656.758,Z 1327.330,A 0.000,B 0.000,C 90.000,E1 95.391} C_DIS
LIN {X -0.202,Y -653.479,Z 1327.327,A 0.000,B 0.000,C 90.000,E1 94.935} C_DIS
LIN {X -0.023,Y -648.972,Z 1327.324,A 0.000,B 0.000,C 90.000,E1 94.302} C_DIS
LIN {X 0.229,Y -645.176,Z 1327.321,A 0.000,B 0.000,C 90.000,E1 93.784} C_DIS
LIN {X -0.225,Y -641.072,Z 1327.318,A 0.000,B 0.000,C 90.000,E1 93.326} C_DIS
LIN {X -0.028,Y -636.609,Z 1327.316,A 0.000,B 0.000,C 90.000,E1 92.808} C_DIS
LIN {X -0.038,Y -629.229,Z 1327.312,A 0.000,B 0.000,C 90.000,E1 92.064} C_DIS
LIN {X 0.134,Y -622.894,Z 1327.308,A 0.000,B 0.000,C 90.000,E1 91.432} C_DIS
LIN {X 0.000,Y -616.564,Z 1327.305,A 0.000,B 0.000,C 90.000,E1 90.859} C_DIS
LIN {X 0.039,Y -609.373,Z 1327.302,A 0.000,B 0.000,C 90.000,E1 90.286} C_DIS
LIN {X 0.014,Y -602.730,Z 1327.299,A 0.000,B 0.000,C 90.000,E1 89.885} C_DIS
LIN {X -0.019,Y -596.088,Z 1327.297,A 0.000,B 0.000,C 90.000,E1 89.542} C_DIS
LIN {X -0.252,Y -589.018,Z 1327.296,A 0.000,B 0.000,C 90.000,E1 89.255} C_DIS
LIN {X 0.180,Y -577.224,Z 1327.293,A 0.000,B 0.000,C 90.000,E1 88.740} C_DIS
LIN {X -0.027,Y -575.175,Z 1327.292,A 0.000,B 0.000,C 90.000,E1 88.625} C_DIS
LIN {X 0.041,Y -573.070,Z 1327.292,A 0.000,B 0.000,C 90.000,E1 88.453} C_DIS
LIN {X 0.270,Y -572.784,Z 1327.291,A 0.000,B 0.000,C 90.000,E1 88.396} C_DIS
LIN {X 0.236,Y -572.762,Z 1327.291,A 0.000,B 0.000,C 90.000,E1 88.396} C_DIS
LIN {X 0.221,Y -571.985,Z 1327.290,A 0.000,B 0.000,C 90.000,E1 88.108} C_DIS
LIN {X -0.076,Y -571.942,Z 1327.287,A 0.000,B 0.000,C 90.000,E1 87.593} C_DIS
LIN {X 0.110,Y -574.159,Z 1327.273,A 0.000,B 0.000,C 90.000,E1 85.122} C_DIS
LIN {X -0.158,Y -576.963,Z 1327.259,A 0.000,B 0.000,C 90.000,E1 82.704} C_DIS
LIN {X 0.028,Y -578.280,Z 1327.253,A 0.000,B 0.000,C 90.000,E1 81.602} C_DIS
LIN {X 0.237,Y -580.512,Z 1327.243,A 0.000,B 0.000,C 90.000,E1 79.690} C_DIS
LIN {X 0.242,Y -582.003,Z 1327.235,A 0.000,B 0.000,C 90.000,E1 78.342} C_DIS
LIN {X 0.279,Y -583.221,Z 1327.228,A 0.000,B 0.000,C 90.000,E1 76.992} C_DIS
LIN {X -0.238,Y -584.328,Z 1327.220,A 0.000,B 0.000,C 90.000,E1 75.700} C_DIS
LIN {X 0.036,Y -585.614,Z 1327.210,A 0.000,B 0.000,C 90.000,E1 73.795} C_DIS
LIN {X 0.021,Y -586.352,Z 1327.204,A 0.000,B 0.000,C 90.000,E1 72.725} C_DIS
LIN {X -0.053,Y -587.568,Z 1327.194,A 0.000,B 0.000,C 90.000,E1 70.859} C_DIS
LIN {X 0.327,Y -588.175,Z 1327.188,A 0.000,B 0.000,C 90.000,E1 69.752} C_DIS
LIN {X -0.067,Y -589.436,Z 1327.177,A 0.000,B 0.000,C 90.000,E1 67.922} C_DIS
LIN {X 0.113,Y -590.464,Z 1327.168,A 0.000,B 0.000,C 90.000,E1 66.305} C_DIS
LIN {X 0.022,Y -591.591,Z 1327.160,A 0.000,B 0.000,C 90.000,E1 64.717} C_DIS
LIN {X -0.041,Y -592.753,Z 1327.151,A 0.000,B 0.000,C 90.000,E1 63.127} C_DIS
LIN {X -0.007,Y -594.488,Z 1327.139,A 0.000,B 0.000,C 90.000,E1 61.001} C_DIS
LIN {X 0.229,Y -596.281,Z 1327.129,A 0.000,B 0.000,C 90.000,E1 59.125} C_DIS
LIN {X -0.213,Y -597.891,Z 1327.120,A 0.000,B 0.000,C 90.000,E1 57.582} C_DIS
LIN {X 0.291,Y -599.311,Z 1327.113,A 0.000,B 0.000,C 90.000,E1 56.215} C_DIS
LIN {X -0.272,Y -600.956,Z 1327.104,A 0.000,B 0.000,C 90.000,E1 54.689} C_DIS
LIN {X 0.132,Y -602.152,Z 1327.096,A 0.000,B 0.000,C 90.000,E1 53.336} C_DIS
LIN {X 0.302,Y -603.123,Z 1327.091,A 0.000,B 0.000,C 90.000,E1 52.271} C_DIS
LIN {X 0.002,Y -603.894,Z 1327.085,A 0.000,B 0.000,C 90.000,E1 51.251} C_DIS
LIN {X 0.353,Y -604.786,Z 1327.078,A 0.000,B 0.000,C 90.000,E1 49.908} C_DIS
LIN {X -0.393,Y -605.305,Z 1327.072,A 0.000,B 0.000,C 90.000,E1 48.933} C_DIS
LIN {X 0.123,Y -605.616,Z 1327.066,A 0.000,B 0.000,C 90.000,E1 47.838} C_DIS
LIN {X -0.348,Y -605.899,Z 1327.056,A 0.000,B 0.000,C 90.000,E1 46.053} C_DIS
LIN {X -0.259,Y -605.913,Z 1327.050,A 0.000,B 0.000,C 90.000,E1 45.000} C_DIS
LIN {X 0.023,Y -605.789,Z 1327.046,A 0.000,B 0.000,C 90.000,E1 44.190} C_DIS
LIN {X 0.156,Y -605.263,Z 1327.037,A 0.000,B 0.000,C 90.000,E1 42.609} C_DIS
LIN {X 0.069,Y -604.821,Z 1327.030,A 0.000,B 0.000,C 90.000,E1 41.310} C_DIS
LIN {X 0.177,Y -604.399,Z 1327.024,A 0.000,B 0.000,C 90.000,E1 40.253} C_DIS
LIN {X -0.013,Y -603.339,Z 1327.012,A 0.000,B 0.000,C 90.000,E1 38.177} C_DIS
LIN {X 0.023,Y -603.010,Z 1327.009,A 0.000,B 0.000,C 90.000,E1 37.649} C_DIS
LIN {X -0.056,Y -602.254,Z 1327.005,A 0.000,B 0.000,C 90.000,E1 36.870} C_DIS
LIN {X 0.111,Y -600.924,Z 1326.999,A 0.000,B 0.000,C 90.000,E1 35.804} C_DIS
LIN {X -0.232,Y -600.113,Z 1326.996,A 0.000,B 0.000,C 90.000,E1 35.311} C_DIS
LIN {X -0.102,Y -598.366,Z 1326.990,A 0.000,B 0.000,C 90.000,E1 34.246} C_DIS
LIN {X 0.161,Y -596.219,Z 1326.984,A 0.000,B 0.000,C 90.000,E1 33.166} C_DIS
LIN {X -0.317,Y -594.387,Z 1326.980,A 0.000,B 0.000,C 90.000,E1 32.418} C_DIS
LIN {X 0.003,Y -592.252,Z 1326.976,A 0.000,B 0.000,C 90.000,E1 31.592} C_DIS
LIN {X -0.013,Y -589.765,Z 1326.971,A 0.000,B 0.000,C 90.000,E1 30.797} C_DIS
LIN {X -0.049,Y -587.049,Z 1326.967,A 0.000,B 0.000,C 90.000,E1 30.001} C_DIS
LIN {X -0.117,Y -583.862,Z 1326.962,A 0.000,B 0.000,C 90.000,E1 29.205} C_DIS
LIN {X 0.357,Y -580.931,Z 1326.958,A 0.000,B 0.000,C 90.000,E1 28.487} C_DIS
LIN {X 0.015,Y -577.726,Z 1326.955,A 0.000,B 0.000,C 90.000,E1 27.847} C_DIS
LIN {X -0.010,Y -574.918,Z 1326.952,A 0.000,B 0.000,C 90.000,E1 27.308} C_DIS
LIN {X 0.191,Y -571.925,Z 1326.949,A 0.000,B 0.000,C 90.000,E1 26.744} C_DIS
LIN {X -0.223,Y -567.881,Z 1326.945,A 0.000,B 0.000,C 90.000,E1 26.104} C_DIS
LIN {X -0.155,Y -563.522,Z 1326.941,A 0.000,B 0.000,C 90.000,E1 25.412} C_DIS
LIN {X -0.027,Y -559.857,Z 1326.938,A 0.000,B 0.000,C 90.000,E1 24.847} C_DIS
LIN {X -0.320,Y -551.625,Z 1326.932,A 0.000,B 0.000,C 90.000,E1 23.770} C_DIS
LIN {X 0.106,Y -545.905,Z 1326.928,A 0.000,B 0.000,C 90.000,E1 23.025} C_DIS
LIN {X 0.205,Y -537.408,Z 1326.922,A 0.000,B 0.000,C 90.000,E1 22.025} C_DIS
LIN {X -0.317,Y -532.544,Z 1326.920,A 0.000,B 0.000,C 90.000,E1 21.535} C_DIS
LIN {X -0.129,Y -522.363,Z 1326.913,A 0.000,B 0.000,C 90.000,E1 20.429} C_DIS
LIN {X -0.118,Y -513.108,Z 1326.908,A 0.000,B 0.000,C 90.000,E1 19.450} C_DIS
LIN {X -0.117,Y -502.486,Z 1326.902,A 0.000,B 0.000,C 90.000,E1 18.362} C_DIS
LIN {X 0.002,Y -492.810,Z 1326.897,A 0.000,B 0.000,C 90.000,E1 17.402} C_DIS
LIN {X 0.050,Y -480.395,Z 1326.890,A 0.000,B 0.000,C 90.000,E1 16.205} C_DIS
LIN {X -0.181,Y -473.164,Z 1326.886,A 0.000,B 0.000,C 90.000,E1 15.552} C_DIS
LIN {X -0.015,Y -458.570,Z 1326.879,A 0.000,B 0.000,C 90.000,E1 14.175} C_DIS
LIN {X -0.073,Y -436.928,Z 1326.867,A 0.000,B 0.000,C 90.000,E1 12.063} C_DIS
LIN {X 0.007,Y -418.401,Z 1326.856,A 0.000,B 0.000,C 90.000,E1 10.074} C_DIS
LIN {X -0.166,Y -404.111,Z 1326.847,A 0.000,B 0.000,C 90.000,E1 8.511} C_DIS
LIN {X 0.097,Y -399.855,Z 1326.844,A 0.000,B 0.000,C 90.000,E1 7.992} C_DIS
LIN {X -0.152,Y -395.329,Z 1326.841,A 0.000,B 0.000,C 90.000,E1 7.409} C_DIS
LIN {X 0.202,Y -395.344,Z 1326.841,A 0.000,B 0.000,C 90.000,E1 7.352} C_DIS
LIN {X -0.075,Y -395.898,Z 1326.840,A 0.000,B 0.000,C 90.000,E1 7.239} C_DIS
LIN {X -0.114,Y -395.923,Z 1326.840,A 0.000,B 0.000,C 90.000,E1 7.239} C_DIS
LIN {X 0.120,Y -399.376,Z 1326.838,A 0.000,B 0.000,C 90.000,E1 6.891} C_DIS
LIN {X -0.171,Y -406.868,Z 1326.836,A 0.000,B 0.000,C 90.000,E1 6.429} C_DIS
LIN {X 0.160,Y -415.134,Z 1326.833,A 0.000,B 0.000,C 90.000,E1 5.853} C_DIS
LIN {X 0.198,Y -416.816,Z 1326.832,A 0.000,B 0.000,C 90.000,E1 5.739} C_DIS
LIN {X -0.185,Y -422.988,Z 1326.830,A 0.000,B 0.000,C 90.000,E1 5.334} C_DIS
LIN {X -0.031,Y -429.111,Z 1326.827,A 0.000,B 0.000,C 90.000,E1 4.821} C_DIS
LIN {X -0.229,Y -436.524,Z 1326.823,A 0.000,B 0.000,C 90.000,E1 4.188} C_DIS
LIN {X -0.040,Y -442.434,Z 1326.820,A 0.000,B 0.000,C 90.000,E1 3.612} C_DIS
LIN {X 0.205,Y -449.514,Z 1326.816,A 0.000,B 0.000,C 90.000,E1 2.865} C_DIS
LIN {X 0.046,Y -455.170,Z 1326.813,A 0.000,B 0.000,C 90.000,E1 2.293} C_DIS
LIN {X -0.086,Y -461.826,Z 1326.809,A 0.000,B 0.000,C 90.000,E1 1.547} C_DIS
LIN {X 0.087,Y -466.883,Z 1326.805,A 0.000,B 0.000,C 90.000,E1 0.917} C_DIS
LIN {X -0.101,Y -472.758,Z 1326.801,A 0.000,B 0.000,C 90.000,E1 0.172} C_DIS
LIN {X 0.103,Y -478.562,Z 1326.796,A 0.000,B 0.000,C 90.000,E1 359.312} C_DIS
LIN {X -0.150,Y -483.525,Z 1326.792,A 0.000,B 0.000,C 90.000,E1 358.568} C_DIS
LIN {X -0.026,Y -489.849,Z 1326.786,A 0.000,B 0.000,C 90.000,E1 357.478} C_DIS
LIN {X 0.141,Y -493.193,Z 1326.783,A 0.000,B 0.000,C 90.000,E1 356.849} C_DIS
LIN {X -0.134,Y -496.318,Z 1326.779,A 0.000,B 0.000,C 90.000,E1 356.274} C_DIS
LIN {X -0.206,Y -499.937,Z 1326.775,A 0.000,B 0.000,C 90.000,E1 355.527} C_DIS
LIN {X -0.244,Y -503.377,Z 1326.771,A 0.000,B 0.000,C 90.000,E1 354.780} C_DIS
LIN {X 0.058,Y -505.922,Z 1326.768,A 0.000,B 0.000,C 90.000,E1 354.147} C_DIS
LIN {X 0.130,Y -508.872,Z 1326.763,A 0.000,B 0.000,C 90.000,E1 353.394} C_DIS
LIN {X -0.183,Y -513.286,Z 1326.757,A 0.000,B 0.000,C 90.000,E1 352.243} C_DIS
LIN {X 0.264,Y -515.223,Z 1326.754,A 0.000,B 0.000,C 90.000,E1 351.602} C_DIS
LIN {X 0.109,Y -518.681,Z 1326.747,A 0.000,B 0.000,C 90.000,E1 350.443} C_DIS
LIN {X 0.092,Y -521.082,Z 1326.742,A 0.000,B 0.000,C 90.000,E1 349.567} C_DIS
LIN {X 0.002,Y -523.118,Z 1326.737,A 0.000,B 0.000,C 90.000,E1 348.701} C_DIS
LIN {X 0.030,Y -524.996,Z 1326.732,A 0.000,B 0.000,C 90.000,E1 347.825} C_DIS
LIN {X 0.193,Y -526.640,Z 1326.728,A 0.000,B 0.000,C 90.000,E1 346.937} C_DIS
LIN {X -0.256,Y -528.059,Z 1326.723,A 0.000,B 0.000,C 90.000,E1 346.117} C_DIS
LIN {X -0.052,Y -529.202,Z 1326.718,A 0.000,B 0.000,C 90.000,E1 345.227} C_DIS
LIN {X 0.166,Y -530.196,Z 1326.713,A 0.000,B 0.000,C 90.000,E1 344.338} C_DIS
LIN {X -0.117,Y -530.882,Z 1326.708,A 0.000,B 0.000,C 90.000,E1 343.504} C_DIS
LIN {X 0.271,Y -531.355,Z 1326.703,A 0.000,B 0.000,C 90.000,E1 342.598} C_DIS
LIN {X -0.002,Y -531.501,Z 1326.699,A 0.000,B 0.000,C 90.000,E1 341.764} C_DIS
LIN {X -0.300,Y -531.437,Z 1326.696,A 0.000,B 0.000,C 90.000,E1 341.221} C_DIS
LIN {X 0.094,Y -531.183,Z 1326.691,A 0.000,B 0.000,C 90.000,E1 340.315} C_DIS
LIN {X 0.169,Y -530.297,Z 1326.684,A 0.000,B 0.000,C 90.000,E1 339.156} C_DIS
LIN {X 0.237,Y -529.170,Z 1326.680,A 0.000,B 0.000,C 90.000,E1 338.284} C_DIS
LIN {X -0.210,Y -527.200,Z 1326.673,A 0.000,B 0.000,C 90.000,E1 337.177} C_DIS
LIN {X 0.140,Y -526.194,Z 1326.670,A 0.000,B 0.000,C 90.000,E1 336.561} C_DIS
LIN {X -0.001,Y -524.944,Z 1326.667,A 0.000,B 0.000,C 90.000,E1 335.997} C_DIS
LIN {X 0.227,Y -522.716,Z 1326.662,A 0.000,B 0.000,C 90.000,E1 335.101} C_DIS
LIN {X 0.253,Y -518.214,Z 1326.654,A 0.000,B 0.000,C 90.000,E1 333.640} C_DIS
LIN {X 0.074,Y -514.524,Z 1326.647,A 0.000,B 0.000,C 90.000,E1 332.487} C_DIS
LIN {X -0.271,Y -509.811,Z 1326.639,A 0.000,B 0.000,C 90.000,E1 331.051} C_DIS
LIN {X 0.108,Y -505.864,Z 1326.632,A 0.000,B 0.000,C 90.000,E1 329.822} C_DIS
LIN {X -0.125,Y -503.685,Z 1326.629,A 0.000,B 0.000,C 90.000,E1 329.253} C_DIS
LIN {X -0.195,Y -500.921,Z 1326.626,A 0.000,B 0.000,C 90.000,E1 328.663} C_DIS
LIN {X -0.027,Y -497.716,Z 1326.622,A 0.000,B 0.000,C 90.000,E1 328.043} C_DIS
LIN {X -0.006,Y -495.820,Z 1326.621,A 0.000,B 0.000,C 90.000,E1 327.740} C_DIS
LIN {X -0.148,Y -493.556,Z 1326.619,A 0.000,B 0.000,C 90.000,E1 327.454} C_DIS
LIN {X -0.088,Y -492.083,Z 1326.618,A 0.000,B 0.000,C 90.000,E1 327.296} C_DIS
LIN {X 0.245,Y -465.745,Z 1326.607,A 0.000,B 0.000,C 90.000,E1 325.182} C_DIS
LIN {X 0.152,Y -443.525,Z 1326.596,A 0.000,B 0.000,C 90.000,E1 323.210} C_DIS
LIN {X 0.216,Y -423.335,Z 1326.584,A 0.000,B 0.000,C 90.000,E1 321.170} C_DIS
LIN {X -0.018,Y -403.746,Z 1326.572,A 0.000,B 0.000,C 90.000,E1 318.976} C_DIS
LIN {X 0.116,Y -386.220,Z 1326.560,A 0.000,B 0.000,C 90.000,E1 316.701} C_DIS
LIN {X 0.194,Y -379.383,Z 1326.554,A 0.000,B 0.000,C 90.000,E1 315.729} C_DIS
LIN {X 0.158,Y -379.362,Z 1326.554,A 0.000,B 0.000,C 90.000,E1 315.729} C_DIS
LIN {X -0.029,Y -384.738,Z 1326.527,A 0.000,B 0.000,C 90.000,E1 310.943} C_DIS
LIN {X 0.214,Y -390.904,Z 1326.494,A 0.000,B 0.000,C 90.000,E1 304.818} C_DIS
LIN {X 0.060,Y -391.345,Z 1326.492,A 0.000,B 0.000,C 90.000,E1 304.485} C_DIS
LIN {X -0.118,Y -397.055,Z 1326.458,A 0.000,B 0.000,C 90.000,E1 298.487} C_DIS
LIN {X 0.188,Y -401.447,Z 1326.427,A 0.000,B 0.000,C 90.000,E1 292.823} C_DIS
LIN {X -0.102,Y -401.676,Z 1326.425,A 0.000,B 0.000,C 90.000,E1 292.514} C_DIS
LIN {X -0.072,Y -404.535,Z 1326.396,A 0.000,B 0.000,C 90.000,E1 287.275} C_DIS
LIN {X 0.028,Y -404.763,Z 1326.394,A 0.000,B 0.000,C 90.000,E1 286.913} C_DIS
LIN {X -0.065,Y -406.151,Z 1326.363,A 0.000,B 0.000,C 90.000,E1 281.366} C_DIS
LIN {X 0.039,Y -405.647,Z 1326.334,A 0.000,B 0.000,C 90.000,E1 276.144} C_DIS
LIN {X 0.045,Y -405.627,Z 1326.332,A 0.000,B 0.000,C 90.000,E1 275.796} C_DIS
LIN {X 0.117,Y -403.555,Z 1326.305,A 0.000,B 0.000,C 90.000,E1 270.917} C_DIS
LIN {X 0.052,Y -403.079,Z 1326.301,A 0.000,B 0.000,C 90.000,E1 270.229} C_DIS
LIN {X -0.121,Y -399.026,Z 1326.272,A 0.000,B 0.000,C 90.000,E1 265.008} C_DIS
LIN {X 0.193,Y -398.153,Z 1326.268,A 0.000,B 0.000,C 90.000,E1 264.261} C_DIS
LIN {X 0.050,Y -392.949,Z 1326.241,A 0.000,B 0.000,C 90.000,E1 259.342} C_DIS
LIN {X 0.007,Y -392.515,Z 1326.239,A 0.000,B 0.000,C 90.000,E1 258.993} C_DIS
LIN {X 0.155,Y -386.146,Z 1326.213,A 0.000,B 0.000,C 90.000,E1 254.338} C_DIS
LIN {X 0.115,Y -385.026,Z 1326.207,A 0.000,B 0.000,C 90.000,E1 253.268} C_DIS
LIN {X -0.012,Y -378.161,Z 1326.183,A 0.000,B 0.000,C 90.000,E1 248.954} C_DIS
LIN {X 0.201,Y -375.924,Z 1326.173,A 0.000,B 0.000,C 90.000,E1 247.102} C_DIS
LIN {X -0.178,Y -369.136,Z 1326.151,A 0.000,B 0.000,C 90.000,E1 243.127} C_DIS
LIN {X 0.050,Y -366.286,Z 1326.138,A 0.000,B 0.000,C 90.000,E1 240.873} C_DIS
LIN {X 0.125,Y -358.371,Z 1326.111,A 0.000,B 0.000,C 90.000,E1 236.008} C_DIS
LIN {X 0.176,Y -356.069,Z 1326.101,A 0.000,B 0.000,C 90.000,E1 234.116} C_DIS
LIN {X -0.070,Y -348.975,Z 1326.075,A 0.000,B 0.000,C 90.000,E1 229.585} C_DIS
LIN {X 0.178,Y -348.984,Z 1326.075,A 0.000,B 0.000,C 90.000,E1 229.542} C_DIS
LIN {X -0.180,Y -362.955,Z 1326.062,A 0.000,B 0.000,C 90.000,E1 227.148} C_DIS
LIN {X -0.011,Y -378.474,Z 1326.048,A 0.000,B 0.000,C 90.000,E1 224.717} C_DIS
LIN {X 0.070,Y -395.567,Z 1326.036,A 0.000,B 0.000,C 90.000,E1 222.366} C_DIS
LIN {X -0.021,Y -413.808,Z 1326.023,A 0.000,B 0.000,C 90.000,E1 220.172} C_DIS
LIN {X -0.121,Y -434.082,Z 1326.011,A 0.000,B 0.000,C 90.000,E1 218.016} C_DIS
LIN {X -0.205,Y -442.943,Z 1326.006,A 0.000,B 0.000,C 90.000,E1 217.156} C_DIS
LIN {X -0.199,Y -444.772,Z 1326.005,A 0.000,B 0.000,C 90.000,E1 216.870} C_DIS
LIN {X 0.107,Y -446.071,Z 1326.003,A 0.000,B 0.000,C 90.000,E1 216.503} C_DIS
LIN {X 0.161,Y -447.059,Z 1326.001,A 0.000,B 0.000,C 90.000,E1 216.171} C_DIS
LIN {X 0.180,Y -448.561,Z 1325.998,A 0.000,B 0.000,C 90.000,E1 215.518} C_DIS
LIN {X -0.050,Y -449.652,Z 1325.994,A 0.000,B 0.000,C 90.000,E1 214.898} C_DIS
LIN {X 0.062,Y -450.883,Z 1325.989,A 0.000,B 0.000,C 90.000,E1 213.913} C_DIS
LIN {X -0.177,Y -452.966,Z 1325.978,A 0.000,B 0.000,C 90.000,E1 212.005} C_DIS
LIN {X 0.011,Y -455.096,Z 1325.967,A 0.000,B 0.000,C 90.000,E1 210.050} C_DIS
LIN {X -0.212,Y -458.215,Z 1325.953,A 0.000,B 0.000,C 90.000,E1 207.513} C_DIS
LIN {X -0.248,Y -461.390,Z 1325.940,A 0.000,B 0.000,C 90.000,E1 205.283} C_DIS
LIN {X 0.243,Y -463.296,Z 1325.933,A 0.000,B 0.000,C 90.000,E1 203.951} C_DIS
LIN {X 0.080,Y -465.448,Z 1325.924,A 0.000,B 0.000,C 90.000,E1 202.386} C_DIS
LIN {X -0.168,Y -467.150,Z 1325.917,A 0.000,B 0.000,C 90.000,E1 201.153} C_DIS
LIN {X -0.218,Y -469.580,Z 1325.907,A 0.000,B 0.000,C 90.000,E1 199.268} C_DIS
LIN {X -0.119,Y -471.206,Z 1325.900,A 0.000,B 0.000,C 90.000,E1 198.000} C_DIS
LIN {X -0.181,Y -473.250,Z 1325.891,A 0.000,B 0.000,C 90.000,E1 196.441} C_DIS
LIN {X 0.247,Y -475.177,Z 1325.883,A 0.000,B 0.000,C 90.000,E1 194.828} C_DIS
LIN {X -0.146,Y -477.462,Z 1325.872,A 0.000,B 0.000,C 90.000,E1 193.008} C_DIS
LIN {X -0.162,Y -480.139,Z 1325.860,A 0.000,B 0.000,C 90.000,E1 190.838} C_DIS
LIN {X 0.069,Y -481.982,Z 1325.852,A 0.000,B 0.000,C 90.000,E1 189.265} C_DIS
LIN {X -0.084,Y -483.462,Z 1325.845,A 0.000,B 0.000,C 90.000,E1 188.049} C_DIS
LIN {X 0.128,Y -485.109,Z 1325.836,A 0.000,B 0.000,C 90.000,E1 186.486} C_DIS
LIN {X -0.040,Y -486.303,Z 1325.829,A 0.000,B 0.000,C 90.000,E1 185.277} C_DIS
LIN {X -0.192,Y -487.361,Z 1325.823,A 0.000,B 0.000,C 90.000,E1 184.069} C_DIS
LIN {X -0.052,Y -487.874,Z 1325.819,A 0.000,B 0.000,C 90.000,E1 183.440} C_DIS
LIN {X 0.115,Y -488.798,Z 1325.811,A 0.000,B 0.000,C 90.000,E1 181.892} C_DIS
LIN {X -0.032,Y -489.317,Z 1325.804,A 0.000,B 0.000,C 90.000,E1 180.688} C_DIS
LIN {X -0.183,Y -489.552,Z 1325.797,A 0.000,B 0.000,C 90.000,E1 179.484} C_DIS
LIN {X 0.154,Y -489.592,Z 1325.790,A 0.000,B 0.000,C 90.000,E1 178.224} C_DIS
LIN {X 0.014,Y -489.286,Z 1325.783,A 0.000,B 0.000,C 90.000,E1 177.020} C_DIS
LIN {X 0.035,Y -488.777,Z 1325.778,A 0.000,B 0.000,C 90.000,E1 176.102} C_DIS
LIN {X 0.090,Y -488.076,Z 1325.773,A 0.000,B 0.000,C 90.000,E1 175.179} C_DIS
LIN {X 0.098,Y -487.162,Z 1325.768,A 0.000,B 0.000,C 90.000,E1 174.261} C_DIS
LIN {X 0.143,Y -486.002,Z 1325.763,A 0.000,B 0.000,C 90.000,E1 173.337} C_DIS
LIN {X 0.177,Y -484.650,Z 1325.758,A 0.000,B 0.000,C 90.000,E1 172.413} C_DIS
LIN {X 0.193,Y -482.796,Z 1325.753,A 0.000,B 0.000,C 90.000,E1 171.489} C_DIS
LIN {X 0.182,Y -480.745,Z 1325.748,A 0.000,B 0.000,C 90.000,E1 170.566} C_DIS
LIN {X -0.103,Y -479.033,Z 1325.744,A 0.000,B 0.000,C 90.000,E1 169.982} C_DIS
LIN {X -0.078,Y -476.077,Z 1325.739,A 0.000,B 0.000,C 90.000,E1 169.050} C_DIS
LIN {X -0.231,Y -474.815,Z 1325.737,A 0.000,B 0.000,C 90.000,E1 168.757} C_DIS
LIN {X -0.164,Y -470.440,Z 1325.732,A 0.000,B 0.000,C 90.000,E1 167.813} C_DIS
LIN {X -0.246,Y -464.737,Z 1325.727,A 0.000,B 0.000,C 90.000,E1 166.881} C_DIS
LIN {X -0.172,Y -454.824,Z 1325.718,A 0.000,B 0.000,C 90.000,E1 165.283} C_DIS
LIN {X -0.007,Y -442.907,Z 1325.707,A 0.000,B 0.000,C 90.000,E1 163.323} C_DIS
LIN {X 0.110,Y -438.391,Z 1325.703,A 0.000,B 0.000,C 90.000,E1 162.489} C_DIS
LIN {X -0.053,Y -436.865,Z 1325.701,A 0.000,B 0.000,C 90.000,E1 162.181} C_DIS
LIN {X -0.096,Y -434.977,Z 1325.698,A 0.000,B 0.000,C 90.000,E1 161.692} C_DIS
LIN {X 0.145,Y -434.215,Z 1325.696,A 0.000,B 0.000,C 90.000,E1 161.329} C_DIS
LIN {X -0.169,Y -433.863,Z 1325.695,A 0.000,B 0.000,C 90.000,E1 161.040} C_DIS
LIN {X 0.120,Y -434.350,Z 1325.692,A 0.000,B 0.000,C 90.000,E1 160.604} C_DIS
LIN {X 0.081,Y -434.386,Z 1325.692,A 0.000,B 0.000,C 90.000,E1 160.604} C_DIS
LIN {X -0.123,Y -435.314,Z 1325.692,A 0.000,B 0.000,C 90.000,E1 160.496} C_DIS
LIN {X 0.017,Y -436.878,Z 1325.690,A 0.000,B 0.000,C 90.000,E1 160.188} C_DIS
LIN {X 0.149,Y -441.850,Z 1325.687,A 0.000,B 0.000,C 90.000,E1 159.699} C_DIS
LIN {X 0.184,Y -461.851,Z 1325.678,A 0.000,B 0.000,C 90.000,E1 158.103} C_DIS
LIN {X 0.084,Y -473.962,Z 1325.673,A 0.000,B 0.000,C 90.000,E1 157.177} C_DIS
LIN {X 0.071,Y -483.112,Z 1325.669,A 0.000,B 0.000,C 90.000,E1 156.433} C_DIS
LIN {X 0.030,Y -490.321,Z 1325.666,A 0.000,B 0.000,C 90.000,E1 155.793} C_DIS
LIN {X 0.225,Y -497.361,Z 1325.662,A 0.000,B 0.000,C 90.000,E1 155.101} C_DIS
LIN {X 0.155,Y -505.546,Z 1325.657,A 0.000,B 0.000,C 90.000,E1 154.280} C_DIS
LIN {X 0.000,Y -512.035,Z 1325.653,A 0.000,B 0.000,C 90.000,E1 153.589} C_DIS
LIN {X 0.166,Y -516.954,Z 1325.650,A 0.000,B 0.000,C 90.000,E1 152.999} C_DIS
LIN {X -0.241,Y -520.421,Z 1325.648,A 0.000,B 0.000,C 90.000,E1 152.615} C_DIS
LIN {X -0.192,Y -524.611,Z 1325.645,A 0.000,B 0.000,C 90.000,E1 152.025} C_DIS
LIN {X 0.201,Y -529.096,Z 1325.641,A 0.000,B 0.000,C 90.000,E1 151.257} C_DIS
LIN {X -0.146,Y -532.103,Z 1325.637,A 0.000,B 0.000,C 90.000,E1 150.717} C_DIS
LIN {X -0.153,Y -535.127,Z 1325.633,A 0.000,B 0.000,C 90.000,E1 149.999} C_DIS
LIN {X -0.004,Y -537.864,Z 1325.629,A 0.000,B 0.000,C 90.000,E1 149.125} C_DIS
LIN {X 0.172,Y -539.496,Z 1325.625,A 0.000,B 0.000,C 90.000,E1 148.535} C_DIS
LIN {X -0.090,Y -541.542,Z 1325.621,A 0.000,B 0.000,C 90.000,E1 147.709} C_DIS
LIN {X 0.109,Y -542.734,Z 1325.617,A 0.000,B 0.000,C 90.000,E1 147.120} C_DIS
LIN {X -0.118,Y -544.201,Z 1325.613,A 0.000,B 0.000,C 90.000,E1 146.294} C_DIS
LIN {X -0.022,Y -545.390,Z 1325.608,A 0.000,B 0.000,C 90.000,E1 145.435} C_DIS
LIN {X -0.218,Y -546.354,Z 1325.603,A 0.000,B 0.000,C 90.000,E1 144.609} C_DIS
LIN {X -0.042,Y -547.388,Z 1325.597,A 0.000,B 0.000,C 90.000,E1 143.463} C_DIS
LIN {X -0.088,Y -548.563,Z 1325.588,A 0.000,B 0.000,C 90.000,E1 141.778} C_DIS
LIN {X 0.077,Y -549.784,Z 1325.580,A 0.000,B 0.000,C 90.000,E1 140.356} C_DIS
LIN {X 0.169,Y -550.376,Z 1325.578,A 0.000,B 0.000,C 90.000,E1 139.989} C_DIS
LIN {X -0.067,Y -550.950,Z 1325.577,A 0.000,B 0.000,C 90.000,E1 139.908} C_DIS
LIN {X 0.048,Y -552.139,Z 1325.576,A 0.000,B 0.000,C 90.000,E1 139.585} C_DIS
LIN {X 0.006,Y -552.192,Z 1325.576,A 0.000,B 0.000,C 90.000,E1 139.585} C_DIS
LIN {X 0.193,Y -554.180,Z 1325.575,A 0.000,B 0.000,C 90.000,E1 139.461} C_DIS
LIN {X -0.192,Y -559.876,Z 1325.574,A 0.000,B 0.000,C 90.000,E1 139.299} C_DIS
LIN {X -0.040,Y -565.490,Z 1325.573,A 0.000,B 0.000,C 90.000,E1 139.138} C_DIS
LIN {X -0.130,Y -568.522,Z 1325.573,A 0.000,B 0.000,C 90.000,E1 139.057} C_DIS
LIN {X 0.061,Y -571.373,Z 1325.572,A 0.000,B 0.000,C 90.000,E1 138.933} C_DIS
LIN {X 0.026,Y -574.353,Z 1325.571,A 0.000,B 0.000,C 90.000,E1 138.809} C_DIS
LIN {X 0.092,Y -580.084,Z 1325.569,A 0.000,B 0.000,C 90.000,E1 138.485} C_DIS
LIN {X 0.295,Y -585.967,Z 1325.567,A 0.000,B 0.000,C 90.000,E1 138.081} C_DIS
LIN {X -0.207,Y -589.971,Z 1325.566,A 0.000,B 0.000,C 90.000,E1 137.838} C_DIS
LIN {X -0.139,Y -595.499,Z 1325.563,A 0.000,B 0.000,C 90.000,E1 137.391} C_DIS
LIN {X -0.020,Y -598.062,Z 1325.562,A 0.000,B 0.000,C 90.000,E1 137.148} C_DIS
LIN {X -0.012,Y -601.812,Z 1325.560,A 0.000,B 0.000,C 90.000,E1 136.782} C_DIS
LIN {X 0.372,Y -609.138,Z 1325.556,A 0.000,B 0.000,C 90.000,E1 135.972} C_DIS
LIN {X -0.047,Y -614.617,Z 1325.552,A 0.000,B 0.000,C 90.000,E1 135.364} C_DIS
LIN {X -0.026,Y -619.715,Z 1325.548,A 0.000,B 0.000,C 90.000,E1 134.717} C_DIS
LIN {X -0.023,Y -625.285,Z 1325.544,A 0.000,B 0.000,C 90.000,E1 133.947} C_DIS
LIN {X 0.044,Y -630.629,Z 1325.540,A 0.000,B 0.000,C 90.000,E1 133.176} C_DIS
LIN {X 0.205,Y -634.879,Z 1325.536,A 0.000,B 0.000,C 90.000,E1 132.528} C_DIS
LIN {X -0.234,Y -642.941,Z 1325.529,A 0.000,B 0.000,C 90.000,E1 131.310} C_DIS
LIN {X 0.014,Y -648.473,Z 1325.525,A 0.000,B 0.000,C 90.000,E1 130.415} C_DIS
LIN {X -0.171,Y -653.685,Z 1325.520,A 0.000,B 0.000,C 90.000,E1 129.564} C_DIS
LIN {X -0.238,Y -658.013,Z 1325.516,A 0.000,B 0.000,C 90.000,E1 128.830} C_DIS
LIN {X 0.183,Y -662.697,Z 1325.511,A 0.000,B 0.000,C 90.000,E1 127.935} C_DIS
LIN {X -0.203,Y -666.415,Z 1325.507,A 0.000,B 0.000,C 90.000,E1 127.237} C_DIS
LIN {X -0.126,Y -668.739,Z 1325.504,A 0.000,B 0.000,C 90.000,E1 126.744} C_DIS
LIN {X -0.056,Y -671.873,Z 1325.500,A 0.000,B 0.000,C 90.000,E1 126.011} C_DIS
LIN {X -0.356,Y -674.759,Z 1325.496,A 0.000,B 0.000,C 90.000,E1 125.311} C_DIS
LIN {X -0.225,Y -676.586,Z 1325.493,A 0.000,B 0.000,C 90.000,E1 124.818} C_DIS
LIN {X 0.082,Y -678.997,Z 1325.489,A 0.000,B 0.000,C 90.000,E1 124.072} C_DIS
LIN {X 0.407,Y -681.735,Z 1325.484,A 0.000,B 0.000,C 90.000,E1 123.086} C_DIS
LIN {X -0.174,Y -683.568,Z 1325.480,A 0.000,B 0.000,C 90.000,E1 122.418} C_DIS
LIN {X 0.209,Y -685.166,Z 1325.476,A 0.000,B 0.000,C 90.000,E1 121.671} C_DIS
LIN {X 0.229,Y -687.007,Z 1325.471,A 0.000,B 0.000,C 90.000,E1 120.718} C_DIS
LIN {X 0.291,Y -688.186,Z 1325.467,A 0.000,B 0.000,C 90.000,E1 120.001} C_DIS
LIN {X -0.231,Y -689.121,Z 1325.463,A 0.000,B 0.000,C 90.000,E1 119.333} C_DIS
LIN {X -0.146,Y -689.671,Z 1325.459,A 0.000,B 0.000,C 90.000,E1 118.615} C_DIS
LIN {X -0.055,Y -690.063,Z 1325.455,A 0.000,B 0.000,C 90.000,E1 117.897} C_DIS
LIN {X -0.041,Y -690.298,Z 1325.450,A 0.000,B 0.000,C 90.000,E1 116.950} C_DIS
LIN {X 0.292,Y -690.136,Z 1325.444,A 0.000,B 0.000,C 90.000,E1 115.976} C_DIS
LIN {X 0.080,Y -689.688,Z 1325.441,A 0.000,B 0.000,C 90.000,E1 115.283} C_DIS
LIN {X -0.078,Y -689.058,Z 1325.438,A 0.000,B 0.000,C 90.000,E1 114.823} C_DIS
LIN {X -0.134,Y -688.714,Z 1325.437,A 0.000,B 0.000,C 90.000,E1 114.591} C_DIS
LIN {X 0.326,Y -687.520,Z 1325.434,A 0.000,B 0.000,C 90.000,E1 114.079} C_DIS
LIN {X -0.355,Y -686.655,Z 1325.433,A 0.000,B 0.000,C 90.000,E1 113.898} C_DIS
LIN {X 0.088,Y -684.341,Z 1325.430,A 0.000,B 0.000,C 90.000,E1 113.387} C_DIS
LIN {X 0.195,Y -683.489,Z 1325.429,A 0.000,B 0.000,C 90.000,E1 113.259} C_DIS
LIN {X -0.222,Y -678.675,Z 1325.427,A 0.000,B 0.000,C 90.000,E1 112.823} C_DIS
LIN {X -0.107,Y -677.093,Z 1325.426,A 0.000,B 0.000,C 90.000,E1 112.695} C_DIS
LIN {X 0.194,Y -668.147,Z 1325.424,A 0.000,B 0.000,C 90.000,E1 112.280} C_DIS
LIN {X 0.227,Y -665.986,Z 1325.424,A 0.000,B 0.000,C 90.000,E1 112.206} C_DIS
LIN {X -0.047,Y -658.616,Z 1325.423,A 0.000,B 0.000,C 90.000,E1 112.078} C_DIS
LIN {X 0.139,Y -656.364,Z 1325.422,A 0.000,B 0.000,C 90.000,E1 112.025} C_DIS
LIN {X -0.083,Y -643.943,Z 1325.422,A 0.000,B 0.000,C 90.000,E1 111.897} C_DIS
LIN {X -0.126,Y -642.172,Z 1325.421,A 0.000,B 0.000,C 90.000,E1 111.844} C_DIS
LIN {X -0.165,Y -642.132,Z 1325.421,A 0.000,B 0.000,C 90.000,E1 111.844} C_DIS
LIN {X -0.120,Y -643.146,Z 1325.420,A 0.000,B 0.000,C 90.000,E1 111.642} C_DIS
LIN {X 0.188,Y -649.238,Z 1325.416,A 0.000,B 0.000,C 90.000,E1 110.865} C_DIS
LIN {X 0.265,Y -651.221,Z 1325.415,A 0.000,B 0.000,C 90.000,E1 110.610} C_DIS
LIN {X 0.073,Y -656.112,Z 1325.411,A 0.000,B 0.000,C 90.000,E1 109.885} C_DIS
LIN {X 0.098,Y -659.757,Z 1325.407,A 0.000,B 0.000,C 90.000,E1 109.268} C_DIS
LIN {X -0.070,Y -662.783,Z 1325.404,A 0.000,B 0.000,C 90.000,E1 108.671} C_DIS
LIN {X -0.152,Y -665.979,Z 1325.400,A 0.000,B 0.000,C 90.000,E1 107.946} C_DIS
LIN {X -0.091,Y -669.623,Z 1325.394,A 0.000,B 0.000,C 90.000,E1 106.968} C_DIS
LIN {X -0.169,Y -670.506,Z 1325.393,A 0.000,B 0.000,C 90.000,E1 106.732} C_DIS
LIN {X -0.378,Y -672.695,Z 1325.389,A 0.000,B 0.000,C 90.000,E1 106.024} C_DIS
LIN {X 0.328,Y -674.015,Z 1325.386,A 0.000,B 0.000,C 90.000,E1 105.481} C_DIS
LIN {X 0.106,Y -676.129,Z 1325.381,A 0.000,B 0.000,C 90.000,E1 104.537} C_DIS
LIN {X 0.056,Y -676.633,Z 1325.380,A 0.000,B 0.000,C 90.000,E1 104.300} C_DIS
LIN {X -0.087,Y -677.689,Z 1325.375,A 0.000,B 0.000,C 90.000,E1 103.592} C_DIS
LIN {X -0.176,Y -678.228,Z 1325.373,A 0.000,B 0.000,C 90.000,E1 103.119} C_DIS
LIN {X 0.355,Y -678.606,Z 1325.369,A 0.000,B 0.000,C 90.000,E1 102.355} C_DIS
LIN {X 0.128,Y -678.710,Z 1325.366,A 0.000,B 0.000,C 90.000,E1 101.895} C_DIS
LIN {X 0.044,Y -678.584,Z 1325.364,A 0.000,B 0.000,C 90.000,E1 101.422} C_DIS
LIN {X -0.046,Y -678.263,Z 1325.361,A 0.000,B 0.000,C 90.000,E1 100.950} C_DIS
LIN {X -0.312,Y -677.299,Z 1325.357,A 0.000,B 0.000,C 90.000,E1 100.254} C_DIS
LIN {X 0.250,Y -676.425,Z 1325.354,A 0.000,B 0.000,C 90.000,E1 99.726} C_DIS
LIN {X 0.025,Y -675.365,Z 1325.352,A 0.000,B 0.000,C 90.000,E1 99.265} C_DIS
LIN {X -0.201,Y -673.817,Z 1325.349,A 0.000,B 0.000,C 90.000,E1 98.803} C_DIS
LIN {X 0.158,Y -670.995,Z 1325.345,A 0.000,B 0.000,C 90.000,E1 98.049} C_DIS
LIN {X -0.090,Y -668.855,Z 1325.342,A 0.000,B 0.000,C 90.000,E1 97.587} C_DIS
LIN {X 0.214,Y -665.259,Z 1325.338,A 0.000,B 0.000,C 90.000,E1 96.834} C_DIS
LIN {X 0.017,Y -663.337,Z 1325.336,A 0.000,B 0.000,C 90.000,E1 96.486} C_DIS
LIN {X 0.084,Y -658.323,Z 1325.331,A 0.000,B 0.000,C 90.000,E1 95.625} C_DIS
LIN {X 0.203,Y -653.460,Z 1325.327,A 0.000,B 0.000,C 90.000,E1 94.878} C_DIS
LIN {X -0.267,Y -648.929,Z 1325.324,A 0.000,B 0.000,C 90.000,E1 94.302} C_DIS
LIN {X -0.014,Y -645.077,Z 1325.321,A 0.000,B 0.000,C 90.000,E1 93.784} C_DIS
LIN {X 0.168,Y -640.938,Z 1325.318,A 0.000,B 0.000,C 90.000,E1 93.269} C_DIS
LIN {X -0.277,Y -636.453,Z 1325.316,A 0.000,B 0.000,C 90.000,E1 92.808} C_DIS
LIN {X -0.261,Y -629.097,Z 1325.311,A 0.000,B 0.000,C 90.000,E1 92.064} C_DIS
LIN {X 0.007,Y -624.062,Z 1325.309,A 0.000,B 0.000,C 90.000,E1 91.547} C_DIS
LIN {X 0.239,Y -617.497,Z 1325.305,A 0.000,B 0.000,C 90.000,E1 90.917} C_DIS
LIN {X 0.166,Y -614.671,Z 1325.304,A 0.000,B 0.000,C 90.000,E1 90.688} C_DIS
LIN {X -0.268,Y -608.902,Z 1325.302,A 0.000,B 0.000,C 90.000,E1 90.286} C_DIS
LIN {X -0.240,Y -602.227,Z 1325.299,A 0.000,B 0.000,C 90.000,E1 89.885} C_DIS
LIN {X 0.231,Y -595.362,Z 1325.297,A 0.000,B 0.000,C 90.000,E1 89.484} C_DIS
LIN {X -0.024,Y -588.043,Z 1325.296,A 0.000,B 0.000,C 90.000,E1 89.198} C_DIS
LIN {X -0.033,Y -577.879,Z 1325.293,A 0.000,B 0.000,C 90.000,E1 88.797} C_DIS
LIN {X -0.155,Y -576.441,Z 1325.293,A 0.000,B 0.000,C 90.000,E1 88.740} C_DIS
LIN {X -0.255,Y -573.729,Z 1325.292,A 0.000,B 0.000,C 90.000,E1 88.568} C_DIS
LIN {X 0.252,Y -572.555,Z 1325.291,A 0.000,B 0.000,C 90.000,E1 88.396} C_DIS
LIN {X 0.220,Y -572.542,Z 1325.291,A 0.000,B 0.000,C 90.000,E1 88.396} C_DIS
LIN {X -0.275,Y -571.988,Z 1325.290,A 0.000,B 0.000,C 90.000,E1 88.224} C_DIS
LIN {X 0.099,Y -571.773,Z 1325.289,A 0.000,B 0.000,C 90.000,E1 88.051} C_DIS
LIN {X -0.015,Y -571.768,Z 1325.287,A 0.000,B 0.000,C 90.000,E1 87.650} C_DIS
LIN {X 0.167,Y -573.999,Z 1325.273,A 0.000,B 0.000,C 90.000,E1 85.179} C_DIS
LIN {X -0.104,Y -576.769,Z 1325.260,A 0.000,B 0.000,C 90.000,E1 82.761} C_DIS
LIN {X 0.210,Y -578.399,Z 1325.252,A 0.000,B 0.000,C 90.000,E1 81.376} C_DIS
LIN {X -0.057,Y -580.644,Z 1325.242,A 0.000,B 0.000,C 90.000,E1 79.511} C_DIS
LIN {X 0.176,Y -581.796,Z 1325.236,A 0.000,B 0.000,C 90.000,E1 78.409} C_DIS
LIN {X 0.199,Y -583.052,Z 1325.228,A 0.000,B 0.000,C 90.000,E1 77.061} C_DIS
LIN {X 0.050,Y -584.352,Z 1325.219,A 0.000,B 0.000,C 90.000,E1 75.463} C_DIS
LIN {X -0.074,Y -585.455,Z 1325.210,A 0.000,B 0.000,C 90.000,E1 73.866} C_DIS
LIN {X -0.252,Y -586.360,Z 1325.203,A 0.000,B 0.000,C 90.000,E1 72.543} C_DIS
LIN {X 0.003,Y -587.423,Z 1325.194,A 0.000,B 0.000,C 90.000,E1 70.913} C_DIS
LIN {X 0.053,Y -588.162,Z 1325.187,A 0.000,B 0.000,C 90.000,E1 69.571} C_DIS
LIN {X -0.007,Y -589.271,Z 1325.178,A 0.000,B 0.000,C 90.000,E1 67.975} C_DIS
LIN {X -0.255,Y -590.133,Z 1325.170,A 0.000,B 0.000,C 90.000,E1 66.666} C_DIS
LIN {X -0.059,Y -591.244,Z 1325.161,A 0.000,B 0.000,C 90.000,E1 65.049} C_DIS
LIN {X -0.137,Y -592.381,Z 1325.153,A 0.000,B 0.000,C 90.000,E1 63.461} C_DIS
LIN {X 0.166,Y -594.105,Z 1325.141,A 0.000,B 0.000,C 90.000,E1 61.307} C_DIS
LIN {X 0.100,Y -595.838,Z 1325.130,A 0.000,B 0.000,C 90.000,E1 59.459} C_DIS
LIN {X 0.252,Y -597.201,Z 1325.123,A 0.000,B 0.000,C 90.000,E1 58.122} C_DIS
LIN {X 0.052,Y -599.136,Z 1325.113,A 0.000,B 0.000,C 90.000,E1 56.294} C_DIS
LIN {X 0.318,Y -600.791,Z 1325.104,A 0.000,B 0.000,C 90.000,E1 54.689} C_DIS
LIN {X -0.371,Y -601.773,Z 1325.098,A 0.000,B 0.000,C 90.000,E1 53.703} C_DIS
LIN {X 0.043,Y -602.965,Z 1325.091,A 0.000,B 0.000,C 90.000,E1 52.351} C_DIS
LIN {X -0.260,Y -603.778,Z 1325.085,A 0.000,B 0.000,C 90.000,E1 51.331} C_DIS
LIN {X 0.086,Y -604.664,Z 1325.078,A 0.000,B 0.000,C 90.000,E1 49.989} C_DIS
LIN {X 0.191,Y -605.201,Z 1325.072,A 0.000,B 0.000,C 90.000,E1 48.933} C_DIS
LIN {X -0.150,Y -605.516,Z 1325.066,A 0.000,B 0.000,C 90.000,E1 47.919} C_DIS
LIN {X 0.233,Y -605.800,Z 1325.056,A 0.000,B 0.000,C 90.000,E1 46.053} C_DIS
LIN {X 0.321,Y -605.836,Z 1325.050,A 0.000,B 0.000,C 90.000,E1 45.000} C_DIS
LIN {X -0.255,Y -605.730,Z 1325.046,A 0.000,B 0.000,C 90.000,E1 44.271} C_DIS
LIN {X -0.318,Y -605.103,Z 1325.036,A 0.000,B 0.000,C 90.000,E1 42.447} C_DIS
LIN {X -0.210,Y -604.762,Z 1325.030,A 0.000,B 0.000,C 90.000,E1 41.391} C_DIS
LIN {X -0.305,Y -604.216,Z 1325.023,A 0.000,B 0.000,C 90.000,E1 40.092} C_DIS
LIN {X 0.084,Y -603.308,Z 1325.012,A 0.000,B 0.000,C 90.000,E1 38.222} C_DIS
LIN {X 0.004,Y -602.761,Z 1325.008,A 0.000,B 0.000,C 90.000,E1 37.443} C_DIS
LIN {X 0.178,Y -601.638,Z 1325.002,A 0.000,B 0.000,C 90.000,E1 36.377} C_DIS
LIN {X 0.089,Y -600.589,Z 1324.998,A 0.000,B 0.000,C 90.000,E1 35.598} C_DIS
LIN {X 0.129,Y -598.402,Z 1324.991,A 0.000,B 0.000,C 90.000,E1 34.278} C_DIS
LIN {X 0.000,Y -596.860,Z 1324.986,A 0.000,B 0.000,C 90.000,E1 33.499} C_DIS
LIN {X 0.027,Y -595.091,Z 1324.982,A 0.000,B 0.000,C 90.000,E1 32.704} C_DIS
LIN {X -0.143,Y -593.082,Z 1324.977,A 0.000,B 0.000,C 90.000,E1 31.926} C_DIS
LIN {X -0.044,Y -591.549,Z 1324.974,A 0.000,B 0.000,C 90.000,E1 31.386} C_DIS
LIN {X -0.178,Y -588.145,Z 1324.969,A 0.000,B 0.000,C 90.000,E1 30.335} C_DIS
LIN {X -0.113,Y -586.257,Z 1324.965,A 0.000,B 0.000,C 90.000,E1 29.795} C_DIS
LIN {X 0.193,Y -581.820,Z 1324.960,A 0.000,B 0.000,C 90.000,E1 28.693} C_DIS
LIN {X -0.008,Y -577.306,Z 1324.954,A 0.000,B 0.000,C 90.000,E1 27.769} C_DIS
LIN {X -0.226,Y -575.219,Z 1324.952,A 0.000,B 0.000,C 90.000,E1 27.385} C_DIS
LIN {X -0.021,Y -572.216,Z 1324.949,A 0.000,B 0.000,C 90.000,E1 26.821} C_DIS
LIN {X -0.177,Y -568.190,Z 1324.945,A 0.000,B 0.000,C 90.000,E1 26.155} C_DIS
LIN {X 0.071,Y -565.629,Z 1324.943,A 0.000,B 0.000,C 90.000,E1 25.720} C_DIS
LIN {X -0.083,Y -559.287,Z 1324.938,A 0.000,B 0.000,C 90.000,E1 24.771} C_DIS
LIN {X 0.079,Y -550.888,Z 1324.931,A 0.000,B 0.000,C 90.000,E1 23.643} C_DIS
LIN {X 0.112,Y -546.315,Z 1324.928,A 0.000,B 0.000,C 90.000,E1 23.078} C_DIS
LIN {X 0.063,Y -536.743,Z 1324.922,A 0.000,B 0.000,C 90.000,E1 21.972} C_DIS
LIN {X 0.034,Y -531.568,Z 1324.919,A 0.000,B 0.000,C 90.000,E1 21.408} C_DIS
LIN {X -0.217,Y -522.688,Z 1324.914,A 0.000,B 0.000,C 90.000,E1 20.482} C_DIS
LIN {X 0.270,Y -513.464,Z 1324.908,A 0.000,B 0.000,C 90.000,E1 19.450} C_DIS
LIN {X -0.117,Y -502.886,Z 1324.902,A 0.000,B 0.000,C 90.000,E1 18.417} C_DIS
LIN {X -0.155,Y -493.580,Z 1324.897,A 0.000,B 0.000,C 90.000,E1 17.511} C_DIS
LIN {X 0.163,Y -482.283,Z 1324.891,A 0.000,B 0.000,C 90.000,E1 16.386} C_DIS
LIN {X -0.180,Y -473.641,Z 1324.887,A 0.000,B 0.000,C 90.000,E1 15.607} C_DIS
LIN {X -0.121,Y -458.941,Z 1324.879,A 0.000,B 0.000,C 90.000,E1 14.245} C_DIS
LIN {X -0.027,Y -437.298,Z 1324.867,A 0.000,B 0.000,C 90.000,E1 12.119} C_DIS
LIN {X 0.024,Y -418.766,Z 1324.856,A 0.000,B 0.000,C 90.000,E1 10.141} C_DIS
LIN {X -0.040,Y -404.489,Z 1324.848,A 0.000,B 0.000,C 90.000,E1 8.568} C_DIS
LIN {X -0.137,Y -398.871,Z 1324.844,A 0.000,B 0.000,C 90.000,E1 7.936} C_DIS
LIN {X 0.031,Y -395.295,Z 1324.841,A 0.000,B 0.000,C 90.000,E1 7.409} C_DIS
LIN {X -0.007,Y -395.275,Z 1324.841,A 0.000,B 0.000,C 90.000,E1 7.409} C_DIS
LIN {X -0.134,Y -395.798,Z 1324.840,A 0.000,B 0.000,C 90.000,E1 7.296} C_DIS
LIN {X -0.172,Y -395.828,Z 1324.840,A 0.000,B 0.000,C 90.000,E1 7.296} C_DIS
LIN {X -0.143,Y -398.970,Z 1324.839,A 0.000,B 0.000,C 90.000,E1 7.004} C_DIS
LIN {X -0.126,Y -402.859,Z 1324.837,A 0.000,B 0.000,C 90.000,E1 6.720} C_DIS
LIN {X -0.092,Y -412.705,Z 1324.834,A 0.000,B 0.000,C 90.000,E1 6.087} C_DIS
LIN {X 0.015,Y -416.067,Z 1324.833,A 0.000,B 0.000,C 90.000,E1 5.853} C_DIS
LIN {X 0.074,Y -423.857,Z 1324.829,A 0.000,B 0.000,C 90.000,E1 5.277} C_DIS
LIN {X -0.165,Y -429.994,Z 1324.827,A 0.000,B 0.000,C 90.000,E1 4.816} C_DIS
LIN {X -0.172,Y -438.998,Z 1324.822,A 0.000,B 0.000,C 90.000,E1 4.012} C_DIS
LIN {X 0.180,Y -443.352,Z 1324.820,A 0.000,B 0.000,C 90.000,E1 3.555} C_DIS
LIN {X 0.132,Y -449.176,Z 1324.817,A 0.000,B 0.000,C 90.000,E1 2.980} C_DIS
LIN {X 0.044,Y -454.859,Z 1324.813,A 0.000,B 0.000,C 90.000,E1 2.407} C_DIS
LIN {X -0.045,Y -461.599,Z 1324.809,A 0.000,B 0.000,C 90.000,E1 1.661} C_DIS
LIN {X 0.008,Y -466.872,Z 1324.806,A 0.000,B 0.000,C 90.000,E1 1.031} C_DIS
LIN {X 0.165,Y -472.908,Z 1324.801,A 0.000,B 0.000,C 90.000,E1 0.229} C_DIS
LIN {X 0.108,Y -479.347,Z 1324.796,A 0.000,B 0.000,C 90.000,E1 359.312} C_DIS
LIN {X -0.138,Y -484.311,Z 1324.792,A 0.000,B 0.000,C 90.000,E1 358.568} C_DIS
LIN {X -0.165,Y -489.777,Z 1324.787,A 0.000,B 0.000,C 90.000,E1 357.650} C_DIS
LIN {X 0.001,Y -493.178,Z 1324.783,A 0.000,B 0.000,C 90.000,E1 357.020} C_DIS
LIN {X 0.220,Y -496.371,Z 1324.780,A 0.000,B 0.000,C 90.000,E1 356.388} C_DIS
LIN {X 0.154,Y -500.034,Z 1324.776,A 0.000,B 0.000,C 90.000,E1 355.641} C_DIS
LIN {X -0.194,Y -504.209,Z 1324.771,A 0.000,B 0.000,C 90.000,E1 354.780} C_DIS
LIN {X 0.116,Y -506.760,Z 1324.768,A 0.000,B 0.000,C 90.000,E1 354.147} C_DIS
LIN {X 0.196,Y -509.723,Z 1324.763,A 0.000,B 0.000,C 90.000,E1 353.394} C_DIS
LIN {X -0.067,Y -513.054,Z 1324.759,A 0.000,B 0.000,C 90.000,E1 352.534} C_DIS
LIN {X -0.161,Y -516.081,Z 1324.754,A 0.000,B 0.000,C 90.000,E1 351.659} C_DIS
LIN {X 0.208,Y -519.588,Z 1324.747,A 0.000,B 0.000,C 90.000,E1 350.443} C_DIS
LIN {X 0.107,Y -521.984,Z 1324.742,A 0.000,B 0.000,C 90.000,E1 349.577} C_DIS
LIN {X 0.133,Y -524.737,Z 1324.736,A 0.000,B 0.000,C 90.000,E1 348.409} C_DIS
LIN {X -0.202,Y -527.092,Z 1324.729,A 0.000,B 0.000,C 90.000,E1 347.285} C_DIS
LIN {X -0.130,Y -528.551,Z 1324.724,A 0.000,B 0.000,C 90.000,E1 346.408} C_DIS
LIN {X 0.081,Y -529.857,Z 1324.720,A 0.000,B 0.000,C 90.000,E1 345.519} C_DIS
LIN {X -0.202,Y -530.900,Z 1324.715,A 0.000,B 0.000,C 90.000,E1 344.685} C_DIS
LIN {X -0.139,Y -531.457,Z 1324.712,A 0.000,B 0.000,C 90.000,E1 344.102} C_DIS
LIN {X 0.253,Y -532.043,Z 1324.707,A 0.000,B 0.000,C 90.000,E1 343.196} C_DIS
LIN {X -0.010,Y -532.508,Z 1324.702,A 0.000,B 0.000,C 90.000,E1 342.362} C_DIS
LIN {X -0.107,Y -532.598,Z 1324.697,A 0.000,B 0.000,C 90.000,E1 341.511} C_DIS
LIN {X -0.179,Y -532.215,Z 1324.691,A 0.000,B 0.000,C 90.000,E1 340.369} C_DIS
LIN {X 0.211,Y -531.894,Z 1324.688,A 0.000,B 0.000,C 90.000,E1 339.752} C_DIS
LIN {X -0.084,Y -531.371,Z 1324.684,A 0.000,B 0.000,C 90.000,E1 339.209} C_DIS
LIN {X -0.001,Y -530.217,Z 1324.680,A 0.000,B 0.000,C 90.000,E1 338.337} C_DIS
LIN {X -0.312,Y -529.366,Z 1324.677,A 0.000,B 0.000,C 90.000,E1 337.794} C_DIS
LIN {X 0.110,Y -526.817,Z 1324.668,A 0.000,B 0.000,C 90.000,E1 336.305} C_DIS
LIN {X -0.198,Y -526.174,Z 1324.667,A 0.000,B 0.000,C 90.000,E1 336.049} C_DIS
LIN {X 0.049,Y -523.891,Z 1324.662,A 0.000,B 0.000,C 90.000,E1 335.153} C_DIS
LIN {X -0.127,Y -519.360,Z 1324.654,A 0.000,B 0.000,C 90.000,E1 333.717} C_DIS
LIN {X -0.053,Y -515.647,Z 1324.647,A 0.000,B 0.000,C 90.000,E1 332.538} C_DIS
LIN {X 0.076,Y -510.945,Z 1324.639,A 0.000,B 0.000,C 90.000,E1 331.051} C_DIS
LIN {X 0.031,Y -506.972,Z 1324.633,A 0.000,B 0.000,C 90.000,E1 329.871} C_DIS
LIN {X -0.016,Y -504.968,Z 1324.629,A 0.000,B 0.000,C 90.000,E1 329.282} C_DIS
LIN {X -0.201,Y -501.425,Z 1324.624,A 0.000,B 0.000,C 90.000,E1 328.408} C_DIS
LIN {X -0.028,Y -498.740,Z 1324.621,A 0.000,B 0.000,C 90.000,E1 327.788} C_DIS
LIN {X -0.081,Y -494.902,Z 1324.617,A 0.000,B 0.000,C 90.000,E1 327.041} C_DIS
LIN {X -0.019,Y -492.225,Z 1324.614,A 0.000,B 0.000,C 90.000,E1 326.580} C_DIS
LIN {X -0.169,Y -490.050,Z 1324.613,A 0.000,B 0.000,C 90.000,E1 326.294} C_DIS
LIN {X -0.111,Y -488.615,Z 1324.612,A 0.000,B 0.000,C 90.000,E1 326.135} C_DIS
LIN {X -0.070,Y -464.188,Z 1324.601,A 0.000,B 0.000,C 90.000,E1 324.116} C_DIS
LIN {X 0.008,Y -442.298,Z 1324.589,A 0.000,B 0.000,C 90.000,E1 322.065} C_DIS
LIN {X -0.097,Y -422.437,Z 1324.578,A 0.000,B 0.000,C 90.000,E1 319.989} C_DIS
LIN {X 0.082,Y -403.210,Z 1324.565,A 0.000,B 0.000,C 90.000,E1 317.676} C_DIS
LIN {X -0.012,Y -386.255,Z 1324.552,A 0.000,B 0.000,C 90.000,E1 315.405} C_DIS
LIN {X -0.023,Y -380.439,Z 1324.548,A 0.000,B 0.000,C 90.000,E1 314.555} C_DIS
LIN {X 0.211,Y -380.438,Z 1324.547,A 0.000,B 0.000,C 90.000,E1 314.514} C_DIS
LIN {X -0.082,Y -384.798,Z 1324.527,A 0.000,B 0.000,C 90.000,E1 310.906} C_DIS
LIN {X -0.092,Y -390.967,Z 1324.493,A 0.000,B 0.000,C 90.000,E1 304.818} C_DIS
LIN {X -0.025,Y -391.371,Z 1324.491,A 0.000,B 0.000,C 90.000,E1 304.452} C_DIS
LIN {X 0.052,Y -396.698,Z 1324.460,A 0.000,B 0.000,C 90.000,E1 298.771} C_DIS
LIN {X -0.077,Y -397.078,Z 1324.458,A 0.000,B 0.000,C 90.000,E1 298.437} C_DIS
